LIN {X 0,Y 418.449,Z 234.861,A -85,B 0,C 180,E1 -9996.753,E2 -9996.753} C_VEL
LIN {X 0,Y 418.302,Z 234.881,A -85,B 0,C 180,E1 -9999.674,E2 -9999.674} C_VEL
LIN {X 0,Y 418.316,Z 234.874,A -85,B 0,C 180,E1 -10003.008,E2 -10003.008} C_VEL
LIN {X 0,Y 418.274,Z 234.878,A -85,B 0,C 180,E1 -10006.738,E2 -10006.738} C_VEL
LIN {X 0,Y 418.234,Z 234.89,A -85,B 0,C 180,E1 -10009.793,E2 -10009.793} C_VEL
LIN {X 0,Y 418.195,Z 234.888,A -85,B 0,C 180,E1 -10012.74,E2 -10012.74} C_VEL
LIN {X 0,Y 418.2,Z 234.893,A -85,B 0,C 180,E1 -10015.91,E2 -10015.91} C_VEL
LIN {X 0,Y 418.228,Z 234.884,A -85,B 0,C 180,E1 -10019.166,E2 -10019.166} C_VEL
LIN {X 0,Y 418.22,Z 234.886,A -85,B 0,C 180,E1 -10022.846,E2 -10022.846} C_VEL
LIN {X 0,Y 418.211,Z 234.892,A -85,B 0,C 180,E1 -10026.241,E2 -10026.241} C_VEL
LIN {X 0,Y 418.172,Z 234.891,A -85,B 0,C 180,E1 -10029.692,E2 -10029.692} C_VEL
LIN {X 0,Y 418.184,Z 234.894,A -85,B 0,C 180,E1 -10032.322,E2 -10032.322} C_VEL
LIN {X 0,Y 418.212,Z 234.889,A -85,B 0,C 180,E1 -10035.113,E2 -10035.113} C_VEL
LIN {X 0,Y 418.202,Z 234.887,A -85,B 0,C 180,E1 -10037.769,E2 -10037.769} C_VEL
LIN {X 0,Y 418.22,Z 234.886,A -85,B 0,C 180,E1 -10041.561,E2 -10041.561} C_VEL
LIN {X 0,Y 418.236,Z 234.889,A -85,B 0,C 180,E1 -10045.163,E2 -10045.163} C_VEL
LIN {X 0,Y 418.229,Z 234.887,A -85,B 0,C 180,E1 -10047.476,E2 -10047.476} C_VEL
LIN {X 0,Y 418.248,Z 234.885,A -85,B 0,C 180,E1 -10050.903,E2 -10050.903} C_VEL
LIN {X 0,Y 418.207,Z 234.887,A -85,B 0,C 180,E1 -10054.097,E2 -10054.097} C_VEL
LIN {X 0,Y 418.22,Z 234.891,A -85,B 0,C 180,E1 -10057.268,E2 -10057.268} C_VEL
LIN {X 0,Y 418.279,Z 234.878,A -85,B 0,C 180,E1 -10060.369,E2 -10060.369} C_VEL
LIN {X 0,Y 418.313,Z 234.878,A -85,B 0,C 180,E1 -10063.409,E2 -10063.409} C_VEL
LIN {X 0,Y 418.346,Z 234.87,A -85,B 0,C 180,E1 -10067.004,E2 -10067.004} C_VEL
LIN {X 0,Y 418.325,Z 234.874,A -85,B 0,C 180,E1 -10070.332,E2 -10070.332} C_VEL
LIN {X 0,Y 418.444,Z 234.858,A -85,B 0,C 180,E1 -10073.252,E2 -10073.252} C_VEL
LIN {X 0,Y 418.319,Z 234.873,A -85,B 0,C 180,E1 -10075.185,E2 -10075.185} C_VEL
LIN {X 0,Y 418.54,Z 234.853,A -85,B 0,C 180,E1 -10078.079,E2 -10078.079} C_VEL
LIN {X 0,Y 418.471,Z 234.854,A -85,B 0,C 180,E1 -10080.966,E2 -10080.966} C_VEL
LIN {X 0,Y 418.475,Z 234.854,A -85,B 0,C 180,E1 -10082.892,E2 -10082.892} C_VEL
LIN {X 0,Y 418.478,Z 234.854,A -85,B 0,C 180,E1 -10085.787,E2 -10085.787} C_VEL
LIN {X 0,Y 418.378,Z 234.87,A -85,B 0,C 180,E1 -10088.699,E2 -10088.699} C_VEL
LIN {X 0,Y 418.322,Z 234.872,A -85,B 0,C 180,E1 -10091.634,E2 -10091.634} C_VEL
LIN {X 0,Y 418.312,Z 234.881,A -85,B 0,C 180,E1 -10094.6,E2 -10094.6} C_VEL
LIN {X 0,Y 418.293,Z 234.876,A -85,B 0,C 180,E1 -10097.607,E2 -10097.607} C_VEL
LIN {X 0,Y 418.263,Z 234.885,A -85,B 0,C 180,E1 -10100.665,E2 -10100.665} C_VEL
LIN {X 0,Y 418.272,Z 234.878,A -85,B 0,C 180,E1 -10103.785,E2 -10103.785} C_VEL
LIN {X 0,Y 418.222,Z 234.893,A -85,B 0,C 180,E1 -10107.044,E2 -10107.044} C_VEL
LIN {X 0,Y 418.254,Z 234.881,A -85,B 0,C 180,E1 -10110.274,E2 -10110.274} C_VEL
LIN {X 0,Y 418.248,Z 234.884,A -85,B 0,C 180,E1 -10113.68,E2 -10113.68} C_VEL
LIN {X 0,Y 418.253,Z 234.887,A -85,B 0,C 180,E1 -10117.226,E2 -10117.226} C_VEL
LIN {X 0,Y 418.223,Z 234.886,A -85,B 0,C 180,E1 -10120.868,E2 -10120.868} C_VEL
LIN {X 0,Y 418.218,Z 234.891,A -85,B 0,C 180,E1 -10123.729,E2 -10123.729} C_VEL
LIN {X 0,Y 418.214,Z 234.886,A -85,B 0,C 180,E1 -10126.448,E2 -10126.448} C_VEL
LIN {X 0,Y 418.222,Z 234.886,A -85,B 0,C 180,E1 -10129.133,E2 -10129.133} C_VEL
LIN {X 0,Y 418.253,Z 234.881,A -85,B 0,C 180,E1 -10132.776,E2 -10132.776} C_VEL
LIN {X 0,Y 418.264,Z 234.883,A -85,B 0,C 180,E1 -10136.323,E2 -10136.323} C_VEL
LIN {X 0,Y 418.257,Z 234.883,A -85,B 0,C 180,E1 -10139.728,E2 -10139.728} C_VEL
LIN {X 0,Y 418.259,Z 234.887,A -85,B 0,C 180,E1 -10143.019,E2 -10143.019} C_VEL
LIN {X 0,Y 418.334,Z 234.998,A -85,B 0,C 180,E1 -10143.764,E2 -10143.764} C_VEL
LIN {X 0,Y 420.475,Z 246.2,A -85,B 0,C 180,E1 -10146.349,E2 -10146.349} C_VEL
LIN {X 0,Y 420.71,Z 251.116,A -85,B 0,C 180,E1 -10147.403,E2 -10147.403} C_VEL
LIN {X 0,Y 419.72,Z 266.974,A -85,B 0,C 180,E1 -10150.687,E2 -10150.687} C_VEL
LIN {X 0,Y 419.594,Z 269.57,A -85,B 0,C 180,E1 -10151.165,E2 -10151.165} C_VEL
LIN {X 0,Y 423.421,Z 293.744,A -85,B 0,C 180,E1 -10151.771,E2 -10151.771} C_VEL
LIN {X 0,Y 422.421,Z 377.284,A -85,B 0,C 180,E1 -10153.227,E2 -10153.227} C_VEL
LIN {X 0,Y 421.945,Z 390.495,A -85,B 0,C 180,E1 -10153.643,E2 -10153.643} C_VEL
LIN {X 0,Y 421.367,Z 403.772,A -85,B 0,C 180,E1 -10154.273,E2 -10154.273} C_VEL
LIN {X 0,Y 420.746,Z 414.923,A -85,B 0,C 180,E1 -10154.993,E2 -10154.993} C_VEL
LIN {X 0,Y 420.035,Z 426.239,A -85,B 0,C 180,E1 -10155.93,E2 -10155.93} C_VEL
LIN {X 0,Y 419.34,Z 436.982,A -85,B 0,C 180,E1 -10157.045,E2 -10157.045} C_VEL
LIN {X 0,Y 418.811,Z 445.521,A -85,B 0,C 180,E1 -10158.136,E2 -10158.136} C_VEL
LIN {X 0,Y 418.21,Z 453.382,A -85,B 0,C 180,E1 -10159.346,E2 -10159.346} C_VEL
LIN {X 0,Y 417.745,Z 461.051,A -85,B 0,C 180,E1 -10160.802,E2 -10160.802} C_VEL
LIN {X 0,Y 417.394,Z 467.211,A -85,B 0,C 180,E1 -10162.257,E2 -10162.257} C_VEL
LIN {X 0,Y 417.159,Z 472.14,A -85,B 0,C 180,E1 -10163.728,E2 -10163.728} C_VEL
LIN {X 0,Y 417.119,Z 475.84,A -85,B 0,C 180,E1 -10165.166,E2 -10165.166} C_VEL
LIN {X 0,Y 417.004,Z 477.771,A -85,B 0,C 180,E1 -10166.133,E2 -10166.133} C_VEL
LIN {X 0,Y 416.988,Z 479.275,A -85,B 0,C 180,E1 -10167.1,E2 -10167.1} C_VEL
LIN {X 0,Y 417.034,Z 480.328,A -85,B 0,C 180,E1 -10168.067,E2 -10168.067} C_VEL
LIN {X 0,Y 416.987,Z 481.263,A -85,B 0,C 180,E1 -10169.998,E2 -10169.998} C_VEL
LIN {X 0,Y 416.996,Z 481.142,A -85,B 0,C 180,E1 -10170.964,E2 -10170.964} C_VEL
LIN {X 0,Y 417.034,Z 480.589,A -85,B 0,C 180,E1 -10171.93,E2 -10171.93} C_VEL
LIN {X 0,Y 417.003,Z 478.309,A -85,B 0,C 180,E1 -10173.864,E2 -10173.864} C_VEL
LIN {X 0,Y 417.162,Z 475.485,A -85,B 0,C 180,E1 -10175.315,E2 -10175.315} C_VEL
LIN {X 0,Y 417.25,Z 471.64,A -85,B 0,C 180,E1 -10176.77,E2 -10176.77} C_VEL
LIN {X 0,Y 417.549,Z 466.675,A -85,B 0,C 180,E1 -10178.224,E2 -10178.224} C_VEL
LIN {X 0,Y 417.995,Z 460.442,A -85,B 0,C 180,E1 -10179.678,E2 -10179.678} C_VEL
LIN {X 0,Y 418.561,Z 452.662,A -85,B 0,C 180,E1 -10181.132,E2 -10181.132} C_VEL
LIN {X 0,Y 419.27,Z 444.726,A -85,B 0,C 180,E1 -10182.339,E2 -10182.339} C_VEL
LIN {X 0,Y 420.016,Z 435.055,A -85,B 0,C 180,E1 -10183.546,E2 -10183.546} C_VEL
LIN {X 0,Y 420.753,Z 424.328,A -85,B 0,C 180,E1 -10184.632,E2 -10184.632} C_VEL
LIN {X 0,Y 421.469,Z 413.916,A -85,B 0,C 180,E1 -10185.472,E2 -10185.472} C_VEL
LIN {X 0,Y 422.273,Z 401.439,A -85,B 0,C 180,E1 -10186.247,E2 -10186.247} C_VEL
LIN {X 0,Y 422.89,Z 388.32,A -85,B 0,C 180,E1 -10186.844,E2 -10186.844} C_VEL
LIN {X 0,Y 423.378,Z 376.495,A -85,B 0,C 180,E1 -10187.197,E2 -10187.197} C_VEL
LIN {X 0,Y 424.274,Z 292.712,A -85,B 0,C 180,E1 -10188.681,E2 -10188.681} C_VEL
LIN {X 0,Y 420.613,Z 272.268,A -85,B 0,C 180,E1 -10189.247,E2 -10189.247} C_VEL
LIN {X 0,Y 420.049,Z 269.214,A -85,B 0,C 180,E1 -10189.362,E2 -10189.362} C_VEL
LIN {X 0,Y 421.091,Z 253.587,A -85,B 0,C 180,E1 -10192.572,E2 -10192.572} C_VEL
LIN {X 0,Y 421.085,Z 248.782,A -85,B 0,C 180,E1 -10193.612,E2 -10193.612} C_VEL
LIN {X 0,Y 418.995,Z 238.02,A -85,B 0,C 180,E1 -10196.121,E2 -10196.121} C_VEL
LIN {X 0,Y 418.302,Z 234.921,A -85,B 0,C 180,E1 -10196.941,E2 -10196.941} C_VEL
LIN {X 0,Y 418.248,Z 234.885,A -85,B 0,C 180,E1 -10200.27,E2 -10200.27} C_VEL
LIN {X 0,Y 418.251,Z 234.886,A -85,B 0,C 180,E1 -10203.675,E2 -10203.675} C_VEL
LIN {X 0,Y 418.24,Z 234.886,A -85,B 0,C 180,E1 -10207.222,E2 -10207.222} C_VEL
LIN {X 0,Y 418.234,Z 234.886,A -85,B 0,C 180,E1 -10209.681,E2 -10209.681} C_VEL
LIN {X 0,Y 418.224,Z 234.882,A -85,B 0,C 180,E1 -10212.317,E2 -10212.317} C_VEL
LIN {X 0,Y 418.235,Z 234.883,A -85,B 0,C 180,E1 -10215.106,E2 -10215.106} C_VEL
LIN {X 0,Y 418.232,Z 234.879,A -85,B 0,C 180,E1 -10217.763,E2 -10217.763} C_VEL
LIN {X 0,Y 418.236,Z 234.884,A -85,B 0,C 180,E1 -10221.553,E2 -10221.553} C_VEL
LIN {X 0,Y 418.257,Z 234.884,A -85,B 0,C 180,E1 -10225.156,E2 -10225.156} C_VEL
LIN {X 0,Y 418.243,Z 234.881,A -85,B 0,C 180,E1 -10227.469,E2 -10227.469} C_VEL
LIN {X 0,Y 418.26,Z 234.882,A -85,B 0,C 180,E1 -10230.894,E2 -10230.894} C_VEL
LIN {X 0,Y 418.225,Z 234.885,A -85,B 0,C 180,E1 -10234.09,E2 -10234.09} C_VEL
LIN {X 0,Y 418.222,Z 234.888,A -85,B 0,C 180,E1 -10237.26,E2 -10237.26} C_VEL
LIN {X 0,Y 418.276,Z 234.878,A -85,B 0,C 180,E1 -10240.361,E2 -10240.361} C_VEL
LIN {X 0,Y 418.309,Z 234.874,A -85,B 0,C 180,E1 -10243.401,E2 -10243.401} C_VEL
LIN {X 0,Y 418.337,Z 234.873,A -85,B 0,C 180,E1 -10246.996,E2 -10246.996} C_VEL
LIN {X 0,Y 418.318,Z 234.874,A -85,B 0,C 180,E1 -10250.325,E2 -10250.325} C_VEL
LIN {X 0,Y 418.454,Z 234.856,A -85,B 0,C 180,E1 -10253.245,E2 -10253.245} C_VEL
LIN {X 0,Y 418.304,Z 234.881,A -85,B 0,C 180,E1 -10255.178,E2 -10255.178} C_VEL
LIN {X 0,Y 418.517,Z 234.85,A -85,B 0,C 180,E1 -10258.072,E2 -10258.072} C_VEL
LIN {X 0,Y 418.389,Z 234.864,A -85,B 0,C 180,E1 -10260.959,E2 -10260.959} C_VEL
LIN {X 0,Y 418.456,Z 234.856,A -85,B 0,C 180,E1 -10262.884,E2 -10262.884} C_VEL
LIN {X 0,Y 418.422,Z 234.86,A -85,B 0,C 180,E1 -10266.748,E2 -10266.748} C_VEL
LIN {X 0,Y 418.318,Z 234.874,A -85,B 0,C 180,E1 -10269.668,E2 -10269.668} C_VEL
LIN {X 0,Y 418.325,Z 234.87,A -85,B 0,C 180,E1 -10272.997,E2 -10272.997} C_VEL
LIN {X 0,Y 418.289,Z 234.876,A -85,B 0,C 180,E1 -10276.731,E2 -10276.731} C_VEL
LIN {X 0,Y 418.246,Z 234.885,A -85,B 0,C 180,E1 -10279.786,E2 -10279.786} C_VEL
LIN {X 0,Y 418.205,Z 234.889,A -85,B 0,C 180,E1 -10282.733,E2 -10282.733} C_VEL
LIN {X 0,Y 418.24,Z 234.885,A -85,B 0,C 180,E1 -10285.901,E2 -10285.901} C_VEL
LIN {X 0,Y 418.235,Z 234.88,A -85,B 0,C 180,E1 -10289.159,E2 -10289.159} C_VEL
LIN {X 0,Y 418.226,Z 234.884,A -85,B 0,C 180,E1 -10292.841,E2 -10292.841} C_VEL
LIN {X 0,Y 418.216,Z 234.886,A -85,B 0,C 180,E1 -10296.236,E2 -10296.236} C_VEL
LIN {X 0,Y 418.232,Z 234.888,A -85,B 0,C 180,E1 -10299.677,E2 -10299.677} C_VEL
LIN {X 0,Y 418.249,Z 234.885,A -85,B 0,C 180,E1 -10302.327,E2 -10302.327} C_VEL
LIN {X 0,Y 418.289,Z 234.973,A -85,B 0,C 180,E1 -10304.337,E2 -10304.337} C_VEL
LIN {X 0,Y 419.722,Z 241.882,A -85,B 0,C 180,E1 -10306.048,E2 -10306.048} C_VEL
LIN {X 0,Y 420.664,Z 247.281,A -85,B 0,C 180,E1 -10307.308,E2 -10307.308} C_VEL
LIN {X 0,Y 420.284,Z 256.46,A -85,B 0,C 180,E1 -10309.298,E2 -10309.298} C_VEL
LIN {X 0,Y 420.229,Z 258.615,A -85,B 0,C 180,E1 -10309.697,E2 -10309.697} C_VEL
LIN {X 0,Y 424.167,Z 278.047,A -85,B 0,C 180,E1 -10310.287,E2 -10310.287} C_VEL
LIN {X 0,Y 424.537,Z 281.534,A -85,B 0,C 180,E1 -10310.369,E2 -10310.369} C_VEL
LIN {X 0,Y 423.399,Z 365.98,A -85,B 0,C 180,E1 -10311.858,E2 -10311.858} C_VEL
LIN {X 0,Y 422.926,Z 379.212,A -85,B 0,C 180,E1 -10312.279,E2 -10312.279} C_VEL
LIN {X 0,Y 422.339,Z 391.655,A -85,B 0,C 180,E1 -10312.868,E2 -10312.868} C_VEL
LIN {X 0,Y 421.708,Z 402.839,A -85,B 0,C 180,E1 -10313.581,E2 -10313.581} C_VEL
LIN {X 0,Y 420.896,Z 414.682,A -85,B 0,C 180,E1 -10314.562,E2 -10314.562} C_VEL
LIN {X 0,Y 420.119,Z 424.963,A -85,B 0,C 180,E1 -10315.628,E2 -10315.628} C_VEL
LIN {X 0,Y 419.404,Z 433.62,A -85,B 0,C 180,E1 -10316.727,E2 -10316.727} C_VEL
LIN {X 0,Y 418.702,Z 442.352,A -85,B 0,C 180,E1 -10318.082,E2 -10318.082} C_VEL
LIN {X 0,Y 418.028,Z 450.685,A -85,B 0,C 180,E1 -10319.713,E2 -10319.713} C_VEL
LIN {X 0,Y 417.741,Z 456.001,A -85,B 0,C 180,E1 -10321.014,E2 -10321.014} C_VEL
LIN {X 0,Y 417.405,Z 460.637,A -85,B 0,C 180,E1 -10322.419,E2 -10322.419} C_VEL
LIN {X 0,Y 417.16,Z 464.674,A -85,B 0,C 180,E1 -10324.024,E2 -10324.024} C_VEL
LIN {X 0,Y 416.946,Z 467.333,A -85,B 0,C 180,E1 -10325.522,E2 -10325.522} C_VEL
LIN {X 0,Y 416.8,Z 469.126,A -85,B 0,C 180,E1 -10327.183,E2 -10327.183} C_VEL
LIN {X 0,Y 416.823,Z 469.641,A -85,B 0,C 180,E1 -10328.228,E2 -10328.228} C_VEL
LIN {X 0,Y 416.779,Z 469.681,A -85,B 0,C 180,E1 -10329.263,E2 -10329.263} C_VEL
LIN {X 0,Y 416.874,Z 468.974,A -85,B 0,C 180,E1 -10330.733,E2 -10330.733} C_VEL
LIN {X 0,Y 416.903,Z 467.138,A -85,B 0,C 180,E1 -10332.338,E2 -10332.338} C_VEL
LIN {X 0,Y 417.086,Z 464.431,A -85,B 0,C 180,E1 -10333.813,E2 -10333.813} C_VEL
LIN {X 0,Y 417.278,Z 460.442,A -85,B 0,C 180,E1 -10335.368,E2 -10335.368} C_VEL
LIN {X 0,Y 417.558,Z 455.374,A -85,B 0,C 180,E1 -10336.868,E2 -10336.868} C_VEL
LIN {X 0,Y 417.962,Z 448.983,A -85,B 0,C 180,E1 -10338.361,E2 -10338.361} C_VEL
LIN {X 0,Y 418.45,Z 440.984,A -85,B 0,C 180,E1 -10339.844,E2 -10339.844} C_VEL
LIN {X 0,Y 419.056,Z 432.78,A -85,B 0,C 180,E1 -10341.077,E2 -10341.077} C_VEL
LIN {X 0,Y 419.673,Z 422.808,A -85,B 0,C 180,E1 -10342.302,E2 -10342.302} C_VEL
LIN {X 0,Y 419.733,Z 422.251,A -85,B 0,C 180,E1 -10342.364,E2 -10342.364} C_VEL
LIN {X 0,Y 419.504,Z 417.637,A -85,B 0,C 180,E1 -10342.867,E2 -10342.867} C_VEL
LIN {X 0,Y 417.189,Z 409.926,A -85,B 0,C 180,E1 -10343.663,E2 -10343.663} C_VEL
LIN {X 0,Y 414.801,Z 401.806,A -85,B 0,C 180,E1 -10344.38,E2 -10344.38} C_VEL
LIN {X 0,Y 414.451,Z 396.549,A -85,B 0,C 180,E1 -10344.75,E2 -10344.75} C_VEL
LIN {X 0,Y 414.994,Z 384.483,A -85,B 0,C 180,E1 -10345.412,E2 -10345.412} C_VEL
LIN {X 0,Y 415.503,Z 371.242,A -85,B 0,C 180,E1 -10345.922,E2 -10345.922} C_VEL
LIN {X 0,Y 415.745,Z 357.284,A -85,B 0,C 180,E1 -10346.239,E2 -10346.239} C_VEL
LIN {X 0,Y 416.51,Z 280.026,A -85,B 0,C 180,E1 -10347.584,E2 -10347.584} C_VEL
LIN {X 0,Y 412.836,Z 258.965,A -85,B 0,C 180,E1 -10348.142,E2 -10348.142} C_VEL
LIN {X 0,Y 412.957,Z 255.755,A -85,B 0,C 180,E1 -10348.783,E2 -10348.783} C_VEL
LIN {X 0,Y 413.419,Z 247.118,A -85,B 0,C 180,E1 -10350.732,E2 -10350.732} C_VEL
LIN {X 0,Y 411.82,Z 238.008,A -85,B 0,C 180,E1 -10352.936,E2 -10352.936} C_VEL
LIN {X 0,Y 411.281,Z 235.803,A -85,B 0,C 180,E1 -10353.553,E2 -10353.553} C_VEL
LIN {X 0,Y 411.431,Z 235.736,A -85,B 0,C 180,E1 -10355.884,E2 -10355.884} C_VEL
LIN {X 0,Y 411.314,Z 235.746,A -85,B 0,C 180,E1 -10358.848,E2 -10358.848} C_VEL
LIN {X 0,Y 411.258,Z 235.757,A -85,B 0,C 180,E1 -10361.835,E2 -10361.835} C_VEL
LIN {X 0,Y 411.222,Z 235.757,A -85,B 0,C 180,E1 -10364.855,E2 -10364.855} C_VEL
LIN {X 0,Y 411.214,Z 235.764,A -85,B 0,C 180,E1 -10367.918,E2 -10367.918} C_VEL
LIN {X 0,Y 411.16,Z 235.764,A -85,B 0,C 180,E1 -10371.037,E2 -10371.037} C_VEL
LIN {X 0,Y 411.168,Z 235.768,A -85,B 0,C 180,E1 -10374.22,E2 -10374.22} C_VEL
LIN {X 0,Y 411.154,Z 235.766,A -85,B 0,C 180,E1 -10377.487,E2 -10377.487} C_VEL
LIN {X 0,Y 411.157,Z 235.766,A -85,B 0,C 180,E1 -10380.852,E2 -10380.852} C_VEL
LIN {X 0,Y 411.163,Z 235.772,A -85,B 0,C 180,E1 -10384.339,E2 -10384.339} C_VEL
LIN {X 0,Y 411.158,Z 235.768,A -85,B 0,C 180,E1 -10386.747,E2 -10386.747} C_VEL
LIN {X 0,Y 411.141,Z 235.767,A -85,B 0,C 180,E1 -10389.724,E2 -10389.724} C_VEL
LIN {X 0,Y 411.139,Z 235.769,A -85,B 0,C 180,E1 -10393.14,E2 -10393.14} C_VEL
LIN {X 0,Y 411.142,Z 235.767,A -85,B 0,C 180,E1 -10395.886,E2 -10395.886} C_VEL
LIN {X 0,Y 411.13,Z 235.776,A -85,B 0,C 180,E1 -10398.779,E2 -10398.779} C_VEL
LIN {X 0,Y 411.169,Z 235.763,A -85,B 0,C 180,E1 -10402.03,E2 -10402.03} C_VEL
LIN {X 0,Y 411.188,Z 235.767,A -85,B 0,C 180,E1 -10405.128,E2 -10405.128} C_VEL
LIN {X 0,Y 411.149,Z 235.766,A -85,B 0,C 180,E1 -10408.007,E2 -10408.007} C_VEL
LIN {X 0,Y 411.161,Z 235.77,A -85,B 0,C 180,E1 -10411.411,E2 -10411.411} C_VEL
LIN {X 0,Y 411.179,Z 235.765,A -85,B 0,C 180,E1 -10414.946,E2 -10414.946} C_VEL
LIN {X 0,Y 411.197,Z 235.762,A -85,B 0,C 180,E1 -10417.918,E2 -10417.918} C_VEL
LIN {X 0,Y 411.214,Z 235.76,A -85,B 0,C 180,E1 -10421.056,E2 -10421.056} C_VEL
LIN {X 0,Y 411.248,Z 235.755,A -85,B 0,C 180,E1 -10424.136,E2 -10424.136} C_VEL
LIN {X 0,Y 411.302,Z 235.748,A -85,B 0,C 180,E1 -10427.17,E2 -10427.17} C_VEL
LIN {X 0,Y 411.279,Z 235.753,A -85,B 0,C 180,E1 -10430.165,E2 -10430.165} C_VEL
LIN {X 0,Y 411.393,Z 235.736,A -85,B 0,C 180,E1 -10433.136,E2 -10433.136} C_VEL
LIN {X 0,Y 411.29,Z 235.748,A -85,B 0,C 180,E1 -10435.103,E2 -10435.103} C_VEL
LIN {X 0,Y 411.508,Z 235.728,A -85,B 0,C 180,E1 -10438.046,E2 -10438.046} C_VEL
LIN {X 0,Y 411.436,Z 235.73,A -85,B 0,C 180,E1 -10440.983,E2 -10440.983} C_VEL
LIN {X 0,Y 411.433,Z 235.731,A -85,B 0,C 180,E1 -10442.941,E2 -10442.941} C_VEL
LIN {X 0,Y 411.4,Z 235.737,A -85,B 0,C 180,E1 -10446.872,E2 -10446.872} C_VEL
LIN {X 0,Y 411.291,Z 235.749,A -85,B 0,C 180,E1 -10449.842,E2 -10449.842} C_VEL
LIN {X 0,Y 411.318,Z 235.746,A -85,B 0,C 180,E1 -10453.107,E2 -10453.107} C_VEL
LIN {X 0,Y 411.271,Z 235.756,A -85,B 0,C 180,E1 -10456.891,E2 -10456.891} C_VEL
LIN {X 0,Y 411.245,Z 235.754,A -85,B 0,C 180,E1 -10459.989,E2 -10459.989} C_VEL
LIN {X 0,Y 411.202,Z 235.764,A -85,B 0,C 180,E1 -10463.151,E2 -10463.151} C_VEL
LIN {X 0,Y 411.19,Z 235.762,A -85,B 0,C 180,E1 -10466.387,E2 -10466.387} C_VEL
LIN {X 0,Y 411.21,Z 235.759,A -85,B 0,C 180,E1 -10469.715,E2 -10469.715} C_VEL
LIN {X 0,Y 411.22,Z 235.764,A -85,B 0,C 180,E1 -10473.158,E2 -10473.158} C_VEL
LIN {X 0,Y 411.207,Z 235.759,A -85,B 0,C 180,E1 -10476.553,E2 -10476.553} C_VEL
LIN {X 0,Y 411.185,Z 235.766,A -85,B 0,C 180,E1 -10479.721,E2 -10479.721} C_VEL
LIN {X 0,Y 411.178,Z 235.765,A -85,B 0,C 180,E1 -10483.136,E2 -10483.136} C_VEL
LIN {X 0,Y 411.178,Z 235.767,A -85,B 0,C 180,E1 -10485.883,E2 -10485.883} C_VEL
LIN {X 0,Y 411.162,Z 235.764,A -85,B 0,C 180,E1 -10488.775,E2 -10488.775} C_VEL
LIN {X 0,Y 411.201,Z 235.765,A -85,B 0,C 180,E1 -10492.025,E2 -10492.025} C_VEL
LIN {X 0,Y 411.221,Z 235.761,A -85,B 0,C 180,E1 -10495.666,E2 -10495.666} C_VEL
LIN {X 0,Y 411.204,Z 235.761,A -85,B 0,C 180,E1 -10499.152,E2 -10499.152} C_VEL
LIN {X 0,Y 411.203,Z 235.764,A -85,B 0,C 180,E1 -10502.517,E2 -10502.517} C_VEL
LIN {X 0,Y 411.282,Z 235.896,A -85,B 0,C 180,E1 -10503.554,E2 -10503.554} C_VEL
LIN {X 0,Y 413.537,Z 247.629,A -85,B 0,C 180,E1 -10506.304,E2 -10506.304} C_VEL
LIN {X 0,Y 413.76,Z 252.034,A -85,B 0,C 180,E1 -10507.266,E2 -10507.266} C_VEL
LIN {X 0,Y 412.651,Z 268.883,A -85,B 0,C 180,E1 -10510.795,E2 -10510.795} C_VEL
LIN {X 0,Y 412.738,Z 270.227,A -85,B 0,C 180,E1 -10510.913,E2 -10510.913} C_VEL
LIN {X 0,Y 416.598,Z 295.2,A -85,B 0,C 180,E1 -10511.529,E2 -10511.529} C_VEL
LIN {X 0,Y 415.571,Z 377.135,A -85,B 0,C 180,E1 -10512.974,E2 -10512.974} C_VEL
LIN {X 0,Y 415.098,Z 390.362,A -85,B 0,C 180,E1 -10513.397,E2 -10513.397} C_VEL
LIN {X 0,Y 414.528,Z 403.095,A -85,B 0,C 180,E1 -10514.006,E2 -10514.006} C_VEL
LIN {X 0,Y 413.857,Z 414.407,A -85,B 0,C 180,E1 -10514.738,E2 -10514.738} C_VEL
LIN {X 0,Y 413.066,Z 426.401,A -85,B 0,C 180,E1 -10515.746,E2 -10515.746} C_VEL
LIN {X 0,Y 412.386,Z 436.603,A -85,B 0,C 180,E1 -10516.823,E2 -10516.823} C_VEL
LIN {X 0,Y 411.805,Z 445.188,A -85,B 0,C 180,E1 -10517.931,E2 -10517.931} C_VEL
LIN {X 0,Y 411.19,Z 453.095,A -85,B 0,C 180,E1 -10519.162,E2 -10519.162} C_VEL
LIN {X 0,Y 410.692,Z 460.807,A -85,B 0,C 180,E1 -10520.642,E2 -10520.642} C_VEL
LIN {X 0,Y 410.348,Z 466.996,A -85,B 0,C 180,E1 -10522.123,E2 -10522.123} C_VEL
LIN {X 0,Y 410.057,Z 472.387,A -85,B 0,C 180,E1 -10523.77,E2 -10523.77} C_VEL
LIN {X 0,Y 410.033,Z 475.674,A -85,B 0,C 180,E1 -10525.082,E2 -10525.082} C_VEL
LIN {X 0,Y 409.924,Z 477.616,A -85,B 0,C 180,E1 -10526.066,E2 -10526.066} C_VEL
LIN {X 0,Y 409.886,Z 479.137,A -85,B 0,C 180,E1 -10527.05,E2 -10527.05} C_VEL
LIN {X 0,Y 409.93,Z 480.204,A -85,B 0,C 180,E1 -10528.034,E2 -10528.034} C_VEL
LIN {X 0,Y 409.922,Z 480.875,A -85,B 0,C 180,E1 -10529.016,E2 -10529.016} C_VEL
LIN {X 0,Y 409.91,Z 481.159,A -85,B 0,C 180,E1 -10529.998,E2 -10529.998} C_VEL
LIN {X 0,Y 409.922,Z 481.053,A -85,B 0,C 180,E1 -10530.981,E2 -10530.981} C_VEL
LIN {X 0,Y 409.93,Z 480.515,A -85,B 0,C 180,E1 -10531.963,E2 -10531.963} C_VEL
LIN {X 0,Y 409.925,Z 478.254,A -85,B 0,C 180,E1 -10533.931,E2 -10533.931} C_VEL
LIN {X 0,Y 410.08,Z 475.45,A -85,B 0,C 180,E1 -10535.407,E2 -10535.407} C_VEL
LIN {X 0,Y 410.188,Z 471.625,A -85,B 0,C 180,E1 -10536.887,E2 -10536.887} C_VEL
LIN {X 0,Y 410.498,Z 466.683,A -85,B 0,C 180,E1 -10538.366,E2 -10538.366} C_VEL
LIN {X 0,Y 410.969,Z 460.473,A -85,B 0,C 180,E1 -10539.845,E2 -10539.845} C_VEL
LIN {X 0,Y 411.562,Z 452.748,A -85,B 0,C 180,E1 -10541.324,E2 -10541.324} C_VEL
LIN {X 0,Y 412.46,Z 443.089,A -85,B 0,C 180,E1 -10542.796,E2 -10542.796} C_VEL
LIN {X 0,Y 413.312,Z 432.87,A -85,B 0,C 180,E1 -10544.051,E2 -10544.051} C_VEL
LIN {X 0,Y 414.107,Z 421.887,A -85,B 0,C 180,E1 -10545.124,E2 -10545.124} C_VEL
LIN {X 0,Y 414.879,Z 410.892,A -85,B 0,C 180,E1 -10545.977,E2 -10545.977} C_VEL
LIN {X 0,Y 415.754,Z 398.708,A -85,B 0,C 180,E1 -10546.699,E2 -10546.699} C_VEL
LIN {X 0,Y 416.313,Z 385.939,A -85,B 0,C 180,E1 -10547.245,E2 -10547.245} C_VEL
LIN {X 0,Y 416.776,Z 372.494,A -85,B 0,C 180,E1 -10547.605,E2 -10547.605} C_VEL
LIN {X 0,Y 417.675,Z 293.704,A -85,B 0,C 180,E1 -10549.01,E2 -10549.01} C_VEL
LIN {X 0,Y 414.142,Z 273.998,A -85,B 0,C 180,E1 -10549.57,E2 -10549.57} C_VEL
LIN {X 0,Y 413.187,Z 269.043,A -85,B 0,C 180,E1 -10549.749,E2 -10549.749} C_VEL
LIN {X 0,Y 414.184,Z 254.928,A -85,B 0,C 180,E1 -10552.706,E2 -10552.706} C_VEL
LIN {X 0,Y 414.264,Z 250.697,A -85,B 0,C 180,E1 -10553.632,E2 -10553.632} C_VEL
LIN {X 0,Y 412.025,Z 239.366,A -85,B 0,C 180,E1 -10556.325,E2 -10556.325} C_VEL
LIN {X 0,Y 411.268,Z 235.805,A -85,B 0,C 180,E1 -10557.268,E2 -10557.268} C_VEL
LIN {X 0,Y 411.205,Z 235.768,A -85,B 0,C 180,E1 -10559.71,E2 -10559.71} C_VEL
LIN {X 0,Y 411.211,Z 235.759,A -85,B 0,C 180,E1 -10563.153,E2 -10563.153} C_VEL
LIN {X 0,Y 411.194,Z 235.765,A -85,B 0,C 180,E1 -10566.549,E2 -10566.549} C_VEL
LIN {X 0,Y 411.2,Z 235.763,A -85,B 0,C 180,E1 -10569.722,E2 -10569.722} C_VEL
LIN {X 0,Y 411.171,Z 235.763,A -85,B 0,C 180,E1 -10573.131,E2 -10573.131} C_VEL
LIN {X 0,Y 411.167,Z 235.761,A -85,B 0,C 180,E1 -10575.879,E2 -10575.879} C_VEL
LIN {X 0,Y 411.152,Z 235.771,A -85,B 0,C 180,E1 -10578.771,E2 -10578.771} C_VEL
LIN {X 0,Y 411.184,Z 235.765,A -85,B 0,C 180,E1 -10582.022,E2 -10582.022} C_VEL
LIN {X 0,Y 411.203,Z 235.761,A -85,B 0,C 180,E1 -10585.663,E2 -10585.663} C_VEL
LIN {X 0,Y 411.186,Z 235.764,A -85,B 0,C 180,E1 -10589.149,E2 -10589.149} C_VEL
LIN {X 0,Y 411.179,Z 235.763,A -85,B 0,C 180,E1 -10591.404,E2 -10591.404} C_VEL
LIN {X 0,Y 411.207,Z 235.76,A -85,B 0,C 180,E1 -10594.931,E2 -10594.931} C_VEL
LIN {X 0,Y 411.197,Z 235.759,A -85,B 0,C 180,E1 -10597.91,E2 -10597.91} C_VEL
LIN {X 0,Y 411.212,Z 235.765,A -85,B 0,C 180,E1 -10601.048,E2 -10601.048} C_VEL
LIN {X 0,Y 411.244,Z 235.752,A -85,B 0,C 180,E1 -10604.128,E2 -10604.128} C_VEL
LIN {X 0,Y 411.294,Z 235.748,A -85,B 0,C 180,E1 -10607.162,E2 -10607.162} C_VEL
LIN {X 0,Y 411.271,Z 235.752,A -85,B 0,C 180,E1 -10610.157,E2 -10610.157} C_VEL
LIN {X 0,Y 411.42,Z 235.73,A -85,B 0,C 180,E1 -10613.129,E2 -10613.129} C_VEL
LIN {X 0,Y 411.277,Z 235.755,A -85,B 0,C 180,E1 -10615.095,E2 -10615.095} C_VEL
LIN {X 0,Y 411.486,Z 235.726,A -85,B 0,C 180,E1 -10618.039,E2 -10618.039} C_VEL
LIN {X 0,Y 411.487,Z 235.727,A -85,B 0,C 180,E1 -10621.954,E2 -10621.954} C_VEL
LIN {X 0,Y 411.367,Z 235.738,A -85,B 0,C 180,E1 -10626.479,E2 -10626.479} C_VEL
LIN {X 0,Y 411.299,Z 235.746,A -85,B 0,C 180,E1 -10628.842,E2 -10628.842} C_VEL
LIN {X 0,Y 411.262,Z 235.758,A -85,B 0,C 180,E1 -10631.829,E2 -10631.829} C_VEL
LIN {X 0,Y 411.236,Z 235.757,A -85,B 0,C 180,E1 -10634.849,E2 -10634.849} C_VEL
LIN {X 0,Y 411.221,Z 235.762,A -85,B 0,C 180,E1 -10637.912,E2 -10637.912} C_VEL
LIN {X 0,Y 411.171,Z 235.765,A -85,B 0,C 180,E1 -10641.031,E2 -10641.031} C_VEL
LIN {X 0,Y 411.193,Z 235.767,A -85,B 0,C 180,E1 -10644.212,E2 -10644.212} C_VEL
LIN {X 0,Y 411.23,Z 235.757,A -85,B 0,C 180,E1 -10647.474,E2 -10647.474} C_VEL
LIN {X 0,Y 411.159,Z 235.769,A -85,B 0,C 180,E1 -10650.844,E2 -10650.844} C_VEL
LIN {X 0,Y 411.175,Z 235.77,A -85,B 0,C 180,E1 -10654.33,E2 -10654.33} C_VEL
LIN {X 0,Y 411.171,Z 235.766,A -85,B 0,C 180,E1 -10657.97,E2 -10657.97} C_VEL
LIN {X 0,Y 411.175,Z 235.77,A -85,B 0,C 180,E1 -10661.233,E2 -10661.233} C_VEL
LIN {X 0,Y 411.261,Z 235.913,A -85,B 0,C 180,E1 -10664.047,E2 -10664.047} C_VEL
LIN {X 0,Y 413.371,Z 246.305,A -85,B 0,C 180,E1 -10666.612,E2 -10666.612} C_VEL
LIN {X 0,Y 413.815,Z 250.306,A -85,B 0,C 180,E1 -10667.542,E2 -10667.542} C_VEL
LIN {X 0,Y 413.365,Z 258.584,A -85,B 0,C 180,E1 -10669.299,E2 -10669.299} C_VEL
LIN {X 0,Y 415.393,Z 267.942,A -85,B 0,C 180,E1 -10669.626,E2 -10669.626} C_VEL
LIN {X 0,Y 417.925,Z 281.248,A -85,B 0,C 180,E1 -10670.012,E2 -10670.012} C_VEL
LIN {X 0,Y 416.703,Z 366.578,A -85,B 0,C 180,E1 -10671.546,E2 -10671.546} C_VEL
LIN {X 0,Y 416.195,Z 380.084,A -85,B 0,C 180,E1 -10671.991,E2 -10671.991} C_VEL
LIN {X 0,Y 415.566,Z 393.064,A -85,B 0,C 180,E1 -10672.633,E2 -10672.633} C_VEL
LIN {X 0,Y 414.769,Z 405.479,A -85,B 0,C 180,E1 -10673.477,E2 -10673.477} C_VEL
LIN {X 0,Y 413.911,Z 416.416,A -85,B 0,C 180,E1 -10674.431,E2 -10674.431} C_VEL
LIN {X 0,Y 413.127,Z 426.7,A -85,B 0,C 180,E1 -10675.556,E2 -10675.556} C_VEL
LIN {X 0,Y 412.39,Z 435.254,A -85,B 0,C 180,E1 -10676.703,E2 -10676.703} C_VEL
LIN {X 0,Y 411.667,Z 443.474,A -85,B 0,C 180,E1 -10678.048,E2 -10678.048} C_VEL
LIN {X 0,Y 410.98,Z 451.612,A -85,B 0,C 180,E1 -10679.706,E2 -10679.706} C_VEL
LIN {X 0,Y 410.578,Z 457.912,A -85,B 0,C 180,E1 -10681.363,E2 -10681.363} C_VEL
LIN {X 0,Y 410.247,Z 462.593,A -85,B 0,C 180,E1 -10682.963,E2 -10682.963} C_VEL
LIN {X 0,Y 410.007,Z 466.156,A -85,B 0,C 180,E1 -10684.628,E2 -10684.628} C_VEL
LIN {X 0,Y 409.836,Z 467.818,A -85,B 0,C 180,E1 -10685.699,E2 -10685.699} C_VEL
LIN {X 0,Y 409.743,Z 468.939,A -85,B 0,C 180,E1 -10686.767,E2 -10686.767} C_VEL
LIN {X 0,Y 409.705,Z 469.622,A -85,B 0,C 180,E1 -10687.85,E2 -10687.85} C_VEL
LIN {X 0,Y 409.693,Z 469.837,A -85,B 0,C 180,E1 -10688.887,E2 -10688.887} C_VEL
LIN {X 0,Y 409.773,Z 469.184,A -85,B 0,C 180,E1 -10690.596,E2 -10690.596} C_VEL
LIN {X 0,Y 409.778,Z 467.742,A -85,B 0,C 180,E1 -10692.02,E2 -10692.02} C_VEL
LIN {X 0,Y 409.979,Z 464.859,A -85,B 0,C 180,E1 -10693.712,E2 -10693.712} C_VEL
LIN {X 0,Y 410.156,Z 461.519,A -85,B 0,C 180,E1 -10695.108,E2 -10695.108} C_VEL
LIN {X 0,Y 410.434,Z 456.707,A -85,B 0,C 180,E1 -10696.636,E2 -10696.636} C_VEL
LIN {X 0,Y 410.787,Z 450.607,A -85,B 0,C 180,E1 -10698.154,E2 -10698.154} C_VEL
LIN {X 0,Y 411.281,Z 443.002,A -85,B 0,C 180,E1 -10699.665,E2 -10699.665} C_VEL
LIN {X 0,Y 411.915,Z 435.208,A -85,B 0,C 180,E1 -10700.921,E2 -10700.921} C_VEL
LIN {X 0,Y 412.545,Z 425.768,A -85,B 0,C 180,E1 -10702.169,E2 -10702.169} C_VEL
LIN {X 0,Y 413.335,Z 415.185,A -85,B 0,C 180,E1 -10703.289,E2 -10703.289} C_VEL
LIN {X 0,Y 414.058,Z 403.46,A -85,B 0,C 180,E1 -10704.279,E2 -10704.279} C_VEL
LIN {X 0,Y 414.451,Z 396.549,A -85,B 0,C 180,E1 -10704.75,E2 -10704.75} C_VEL
LIN {X 0,Y 414.131,Z 391.214,A -85,B 0,C 180,E1 -10705.089,E2 -10705.089} C_VEL
LIN {X 0,Y 411.783,Z 382.369,A -85,B 0,C 180,E1 -10705.628,E2 -10705.628} C_VEL
LIN {X 0,Y 409.293,Z 373.334,A -85,B 0,C 180,E1 -10706.077,E2 -10706.077} C_VEL
LIN {X 0,Y 408.733,Z 367.626,A -85,B 0,C 180,E1 -10706.272,E2 -10706.272} C_VEL
LIN {X 0,Y 409.146,Z 335.693,A -85,B 0,C 180,E1 -10706.877,E2 -10706.877} C_VEL
LIN {X 0,Y 409.76,Z 281.107,A -85,B 0,C 180,E1 -10707.843,E2 -10707.843} C_VEL
LIN {X 0,Y 405.884,Z 258.981,A -85,B 0,C 180,E1 -10708.445,E2 -10708.445} C_VEL
LIN {X 0,Y 406.271,Z 252.937,A -85,B 0,C 180,E1 -10709.754,E2 -10709.754} C_VEL
LIN {X 0,Y 406.37,Z 247.602,A -85,B 0,C 180,E1 -10710.992,E2 -10710.992} C_VEL
LIN {X 0,Y 404.885,Z 239.512,A -85,B 0,C 180,E1 -10712.986,E2 -10712.986} C_VEL
LIN {X 0,Y 404.208,Z 236.669,A -85,B 0,C 180,E1 -10713.771,E2 -10713.771} C_VEL
LIN {X 0,Y 404.379,Z 236.615,A -85,B 0,C 180,E1 -10715.987,E2 -10715.987} C_VEL
LIN {X 0,Y 404.251,Z 236.627,A -85,B 0,C 180,E1 -10719.003,E2 -10719.003} C_VEL
LIN {X 0,Y 404.229,Z 236.63,A -85,B 0,C 180,E1 -10722.044,E2 -10722.044} C_VEL
LIN {X 0,Y 404.168,Z 236.637,A -85,B 0,C 180,E1 -10725.121,E2 -10725.121} C_VEL
LIN {X 0,Y 404.172,Z 236.638,A -85,B 0,C 180,E1 -10728.241,E2 -10728.241} C_VEL
LIN {X 0,Y 404.102,Z 236.646,A -85,B 0,C 180,E1 -10731.423,E2 -10731.423} C_VEL
LIN {X 0,Y 404.126,Z 236.642,A -85,B 0,C 180,E1 -10734.67,E2 -10734.67} C_VEL
LIN {X 0,Y 404.096,Z 236.65,A -85,B 0,C 180,E1 -10738.009,E2 -10738.009} C_VEL
LIN {X 0,Y 404.112,Z 236.649,A -85,B 0,C 180,E1 -10740.289,E2 -10740.289} C_VEL
LIN {X 0,Y 404.108,Z 236.645,A -85,B 0,C 180,E1 -10743.817,E2 -10743.817} C_VEL
LIN {X 0,Y 404.103,Z 236.646,A -85,B 0,C 180,E1 -10746.878,E2 -10746.878} C_VEL
LIN {X 0,Y 404.092,Z 236.647,A -85,B 0,C 180,E1 -10750.079,E2 -10750.079} C_VEL
LIN {X 0,Y 404.118,Z 236.644,A -85,B 0,C 180,E1 -10753.086,E2 -10753.086} C_VEL
LIN {X 0,Y 404.123,Z 236.641,A -85,B 0,C 180,E1 -10755.93,E2 -10755.93} C_VEL
LIN {X 0,Y 404.084,Z 236.651,A -85,B 0,C 180,E1 -10758.638,E2 -10758.638} C_VEL
LIN {X 0,Y 404.123,Z 236.642,A -85,B 0,C 180,E1 -10761.5,E2 -10761.5} C_VEL
LIN {X 0,Y 404.159,Z 236.644,A -85,B 0,C 180,E1 -10764.988,E2 -10764.988} C_VEL
LIN {X 0,Y 404.124,Z 236.642,A -85,B 0,C 180,E1 -10768.448,E2 -10768.448} C_VEL
LIN {X 0,Y 404.138,Z 236.643,A -85,B 0,C 180,E1 -10770.867,E2 -10770.867} C_VEL
LIN {X 0,Y 404.144,Z 236.64,A -85,B 0,C 180,E1 -10774.728,E2 -10774.728} C_VEL
LIN {X 0,Y 404.16,Z 236.643,A -85,B 0,C 180,E1 -10777.513,E2 -10777.513} C_VEL
LIN {X 0,Y 404.158,Z 236.637,A -85,B 0,C 180,E1 -10780.712,E2 -10780.712} C_VEL
LIN {X 0,Y 404.217,Z 236.634,A -85,B 0,C 180,E1 -10783.853,E2 -10783.853} C_VEL
LIN {X 0,Y 404.284,Z 236.621,A -85,B 0,C 180,E1 -10786.943,E2 -10786.943} C_VEL
LIN {X 0,Y 404.246,Z 236.631,A -85,B 0,C 180,E1 -10789.992,E2 -10789.992} C_VEL
LIN {X 0,Y 404.344,Z 236.613,A -85,B 0,C 180,E1 -10793.016,E2 -10793.016} C_VEL
LIN {X 0,Y 404.261,Z 236.624,A -85,B 0,C 180,E1 -10795.017,E2 -10795.017} C_VEL
LIN {X 0,Y 404.477,Z 236.604,A -85,B 0,C 180,E1 -10798.012,E2 -10798.012} C_VEL
LIN {X 0,Y 404.402,Z 236.606,A -85,B 0,C 180,E1 -10801,E2 -10801} C_VEL
LIN {X 0,Y 404.367,Z 236.611,A -85,B 0,C 180,E1 -10802.993,E2 -10802.993} C_VEL
LIN {X 0,Y 404.376,Z 236.613,A -85,B 0,C 180,E1 -10805.989,E2 -10805.989} C_VEL
LIN {X 0,Y 404.268,Z 236.624,A -85,B 0,C 180,E1 -10809.005,E2 -10809.005} C_VEL
LIN {X 0,Y 404.266,Z 236.625,A -85,B 0,C 180,E1 -10812.045,E2 -10812.045} C_VEL
LIN {X 0,Y 404.217,Z 236.632,A -85,B 0,C 180,E1 -10815.121,E2 -10815.121} C_VEL
LIN {X 0,Y 404.218,Z 236.631,A -85,B 0,C 180,E1 -10818.241,E2 -10818.241} C_VEL
LIN {X 0,Y 404.152,Z 236.639,A -85,B 0,C 180,E1 -10821.422,E2 -10821.422} C_VEL
LIN {X 0,Y 404.163,Z 236.64,A -85,B 0,C 180,E1 -10824.67,E2 -10824.67} C_VEL
LIN {X 0,Y 404.118,Z 236.642,A -85,B 0,C 180,E1 -10828.009,E2 -10828.009} C_VEL
LIN {X 0,Y 404.158,Z 236.637,A -85,B 0,C 180,E1 -10830.287,E2 -10830.287} C_VEL
LIN {X 0,Y 404.154,Z 236.639,A -85,B 0,C 180,E1 -10833.815,E2 -10833.815} C_VEL
LIN {X 0,Y 404.15,Z 236.64,A -85,B 0,C 180,E1 -10836.876,E2 -10836.876} C_VEL
LIN {X 0,Y 404.133,Z 236.641,A -85,B 0,C 180,E1 -10840.076,E2 -10840.076} C_VEL
LIN {X 0,Y 404.158,Z 236.639,A -85,B 0,C 180,E1 -10843.083,E2 -10843.083} C_VEL
LIN {X 0,Y 404.135,Z 236.644,A -85,B 0,C 180,E1 -10845.923,E2 -10845.923} C_VEL
LIN {X 0,Y 404.117,Z 236.642,A -85,B 0,C 180,E1 -10848.633,E2 -10848.633} C_VEL
LIN {X 0,Y 404.156,Z 236.64,A -85,B 0,C 180,E1 -10851.495,E2 -10851.495} C_VEL
LIN {X 0,Y 404.199,Z 236.631,A -85,B 0,C 180,E1 -10854.984,E2 -10854.984} C_VEL
LIN {X 0,Y 404.155,Z 236.643,A -85,B 0,C 180,E1 -10858.442,E2 -10858.442} C_VEL
LIN {X 0,Y 404.171,Z 236.64,A -85,B 0,C 180,E1 -10860.863,E2 -10860.863} C_VEL
LIN {X 0,Y 404.229,Z 236.764,A -85,B 0,C 180,E1 -10863.333,E2 -10863.333} C_VEL
LIN {X 0,Y 406.665,Z 249.438,A -85,B 0,C 180,E1 -10866.345,E2 -10866.345} C_VEL
LIN {X 0,Y 406.696,Z 254.173,A -85,B 0,C 180,E1 -10867.386,E2 -10867.386} C_VEL
LIN {X 0,Y 405.708,Z 269.101,A -85,B 0,C 180,E1 -10870.552,E2 -10870.552} C_VEL
LIN {X 0,Y 406.119,Z 272.315,A -85,B 0,C 180,E1 -10870.687,E2 -10870.687} C_VEL
LIN {X 0,Y 409.763,Z 296.104,A -85,B 0,C 180,E1 -10871.273,E2 -10871.273} C_VEL
LIN {X 0,Y 408.714,Z 376.597,A -85,B 0,C 180,E1 -10872.712,E2 -10872.712} C_VEL
LIN {X 0,Y 408.225,Z 389.99,A -85,B 0,C 180,E1 -10873.142,E2 -10873.142} C_VEL
LIN {X 0,Y 407.614,Z 403.372,A -85,B 0,C 180,E1 -10873.792,E2 -10873.792} C_VEL
LIN {X 0,Y 406.868,Z 415.383,A -85,B 0,C 180,E1 -10874.597,E2 -10874.597} C_VEL
LIN {X 0,Y 406.064,Z 427.514,A -85,B 0,C 180,E1 -10875.654,E2 -10875.654} C_VEL
LIN {X 0,Y 405.356,Z 437.252,A -85,B 0,C 180,E1 -10876.718,E2 -10876.718} C_VEL
LIN {X 0,Y 404.688,Z 446.542,A -85,B 0,C 180,E1 -10877.97,E2 -10877.97} C_VEL
LIN {X 0,Y 404.003,Z 455.558,A -85,B 0,C 180,E1 -10879.474,E2 -10879.474} C_VEL
LIN {X 0,Y 403.553,Z 462.812,A -85,B 0,C 180,E1 -10880.981,E2 -10880.981} C_VEL
LIN {X 0,Y 403.168,Z 468.583,A -85,B 0,C 180,E1 -10882.486,E2 -10882.486} C_VEL
LIN {X 0,Y 402.95,Z 473.119,A -85,B 0,C 180,E1 -10883.992,E2 -10883.992} C_VEL
LIN {X 0,Y 402.946,Z 475.508,A -85,B 0,C 180,E1 -10884.996,E2 -10884.996} C_VEL
LIN {X 0,Y 402.846,Z 477.461,A -85,B 0,C 180,E1 -10885.997,E2 -10885.997} C_VEL
LIN {X 0,Y 402.789,Z 478.997,A -85,B 0,C 180,E1 -10886.998,E2 -10886.998} C_VEL
LIN {X 0,Y 402.827,Z 480.081,A -85,B 0,C 180,E1 -10887.999,E2 -10887.999} C_VEL
LIN {X 0,Y 402.85,Z 480.762,A -85,B 0,C 180,E1 -10888.999,E2 -10888.999} C_VEL
LIN {X 0,Y 402.85,Z 480.963,A -85,B 0,C 180,E1 -10890.998,E2 -10890.998} C_VEL
LIN {X 0,Y 402.826,Z 480.44,A -85,B 0,C 180,E1 -10891.998,E2 -10891.998} C_VEL
LIN {X 0,Y 402.849,Z 478.2,A -85,B 0,C 180,E1 -10894,E2 -10894} C_VEL
LIN {X 0,Y 402.98,Z 475.421,A -85,B 0,C 180,E1 -10895.503,E2 -10895.503} C_VEL
LIN {X 0,Y 403.114,Z 471.627,A -85,B 0,C 180,E1 -10897.008,E2 -10897.008} C_VEL
LIN {X 0,Y 403.466,Z 466.72,A -85,B 0,C 180,E1 -10898.513,E2 -10898.513} C_VEL
LIN {X 0,Y 403.947,Z 460.555,A -85,B 0,C 180,E1 -10900.018,E2 -10900.018} C_VEL
LIN {X 0,Y 404.59,Z 452.893,A -85,B 0,C 180,E1 -10901.521,E2 -10901.521} C_VEL
LIN {X 0,Y 405.524,Z 443.284,A -85,B 0,C 180,E1 -10903.019,E2 -10903.019} C_VEL
LIN {X 0,Y 406.402,Z 433.607,A -85,B 0,C 180,E1 -10904.238,E2 -10904.238} C_VEL
LIN {X 0,Y 407.156,Z 423.659,A -85,B 0,C 180,E1 -10905.26,E2 -10905.26} C_VEL
LIN {X 0,Y 408.075,Z 411.371,A -85,B 0,C 180,E1 -10906.25,E2 -10906.25} C_VEL
LIN {X 0,Y 409.007,Z 399.346,A -85,B 0,C 180,E1 -10906.983,E2 -10906.983} C_VEL
LIN {X 0,Y 409.583,Z 387.028,A -85,B 0,C 180,E1 -10907.537,E2 -10907.537} C_VEL
LIN {X 0,Y 410.099,Z 374.335,A -85,B 0,C 180,E1 -10907.901,E2 -10907.901} C_VEL
LIN {X 0,Y 411.083,Z 294.87,A -85,B 0,C 180,E1 -10909.347,E2 -10909.347} C_VEL
LIN {X 0,Y 407.984,Z 277.076,A -85,B 0,C 180,E1 -10909.86,E2 -10909.86} C_VEL
LIN {X 0,Y 406.344,Z 268.943,A -85,B 0,C 180,E1 -10910.148,E2 -10910.148} C_VEL
LIN {X 0,Y 407.374,Z 255.066,A -85,B 0,C 180,E1 -10913.107,E2 -10913.107} C_VEL
LIN {X 0,Y 407.287,Z 251.764,A -85,B 0,C 180,E1 -10913.854,E2 -10913.854} C_VEL
LIN {X 0,Y 405.098,Z 240.718,A -85,B 0,C 180,E1 -10916.532,E2 -10916.532} C_VEL
LIN {X 0,Y 404.216,Z 236.69,A -85,B 0,C 180,E1 -10917.61,E2 -10917.61} C_VEL
LIN {X 0,Y 404.15,Z 236.641,A -85,B 0,C 180,E1 -10920.283,E2 -10920.283} C_VEL
LIN {X 0,Y 404.149,Z 236.645,A -85,B 0,C 180,E1 -10923.81,E2 -10923.81} C_VEL
LIN {X 0,Y 404.137,Z 236.643,A -85,B 0,C 180,E1 -10926.872,E2 -10926.872} C_VEL
LIN {X 0,Y 404.15,Z 236.645,A -85,B 0,C 180,E1 -10930.077,E2 -10930.077} C_VEL
LIN {X 0,Y 404.151,Z 236.638,A -85,B 0,C 180,E1 -10933.08,E2 -10933.08} C_VEL
LIN {X 0,Y 404.147,Z 236.634,A -85,B 0,C 180,E1 -10935.923,E2 -10935.923} C_VEL
LIN {X 0,Y 404.108,Z 236.649,A -85,B 0,C 180,E1 -10938.63,E2 -10938.63} C_VEL
LIN {X 0,Y 404.139,Z 236.64,A -85,B 0,C 180,E1 -10941.492,E2 -10941.492} C_VEL
LIN {X 0,Y 404.182,Z 236.638,A -85,B 0,C 180,E1 -10944.981,E2 -10944.981} C_VEL
LIN {X 0,Y 404.139,Z 236.644,A -85,B 0,C 180,E1 -10948.55,E2 -10948.55} C_VEL
LIN {X 0,Y 404.15,Z 236.639,A -85,B 0,C 180,E1 -10950.859,E2 -10950.859} C_VEL
LIN {X 0,Y 404.136,Z 236.641,A -85,B 0,C 180,E1 -10954.227,E2 -10954.227} C_VEL
LIN {X 0,Y 404.161,Z 236.637,A -85,B 0,C 180,E1 -10957.504,E2 -10957.504} C_VEL
LIN {X 0,Y 404.156,Z 236.64,A -85,B 0,C 180,E1 -10960.704,E2 -10960.704} C_VEL
LIN {X 0,Y 404.212,Z 236.628,A -85,B 0,C 180,E1 -10963.844,E2 -10963.844} C_VEL
LIN {X 0,Y 404.275,Z 236.625,A -85,B 0,C 180,E1 -10966.935,E2 -10966.935} C_VEL
LIN {X 0,Y 404.239,Z 236.629,A -85,B 0,C 180,E1 -10969.984,E2 -10969.984} C_VEL
LIN {X 0,Y 404.37,Z 236.607,A -85,B 0,C 180,E1 -10973.008,E2 -10973.008} C_VEL
LIN {X 0,Y 404.25,Z 236.629,A -85,B 0,C 180,E1 -10975.01,E2 -10975.01} C_VEL
LIN {X 0,Y 404.455,Z 236.602,A -85,B 0,C 180,E1 -10978.005,E2 -10978.005} C_VEL
LIN {X 0,Y 404.456,Z 236.602,A -85,B 0,C 180,E1 -10981.988,E2 -10981.988} C_VEL
LIN {X 0,Y 404.32,Z 236.616,A -85,B 0,C 180,E1 -10986.475,E2 -10986.475} C_VEL
LIN {X 0,Y 404.246,Z 236.625,A -85,B 0,C 180,E1 -10988.998,E2 -10988.998} C_VEL
LIN {X 0,Y 404.235,Z 236.631,A -85,B 0,C 180,E1 -10992.038,E2 -10992.038} C_VEL
LIN {X 0,Y 404.182,Z 236.636,A -85,B 0,C 180,E1 -10995.114,E2 -10995.114} C_VEL
LIN {X 0,Y 404.18,Z 236.64,A -85,B 0,C 180,E1 -10998.235,E2 -10998.235} C_VEL
LIN {X 0,Y 404.113,Z 236.645,A -85,B 0,C 180,E1 -11001.416,E2 -11001.416} C_VEL
LIN {X 0,Y 404.147,Z 236.64,A -85,B 0,C 180,E1 -11004.662,E2 -11004.662} C_VEL
LIN {X 0,Y 404.166,Z 236.634,A -85,B 0,C 180,E1 -11007.996,E2 -11007.996} C_VEL
LIN {X 0,Y 404.108,Z 236.645,A -85,B 0,C 180,E1 -11011.555,E2 -11011.555} C_VEL
LIN {X 0,Y 404.153,Z 236.637,A -85,B 0,C 180,E1 -11015.013,E2 -11015.013} C_VEL
LIN {X 0,Y 404.13,Z 236.643,A -85,B 0,C 180,E1 -11018.753,E2 -11018.753} C_VEL
LIN {X 0,Y 404.156,Z 236.643,A -85,B 0,C 180,E1 -11021.608,E2 -11021.608} C_VEL
LIN {X 0,Y 404.163,Z 236.721,A -85,B 0,C 180,E1 -11023.663,E2 -11023.663} C_VEL
LIN {X 0,Y 406.274,Z 246.74,A -85,B 0,C 180,E1 -11026.218,E2 -11026.218} C_VEL
LIN {X 0,Y 406.923,Z 251.57,A -85,B 0,C 180,E1 -11027.372,E2 -11027.372} C_VEL
LIN {X 0,Y 406.543,Z 258.767,A -85,B 0,C 180,E1 -11028.908,E2 -11028.908} C_VEL
LIN {X 0,Y 408.871,Z 269.34,A -85,B 0,C 180,E1 -11029.283,E2 -11029.283} C_VEL
LIN {X 0,Y 411.333,Z 282.953,A -85,B 0,C 180,E1 -11029.681,E2 -11029.681} C_VEL
LIN {X 0,Y 410.055,Z 366.292,A -85,B 0,C 180,E1 -11031.199,E2 -11031.199} C_VEL
LIN {X 0,Y 409.509,Z 379.897,A -85,B 0,C 180,E1 -11031.649,E2 -11031.649} C_VEL
LIN {X 0,Y 408.902,Z 391.818,A -85,B 0,C 180,E1 -11032.235,E2 -11032.235} C_VEL
LIN {X 0,Y 408.227,Z 402.725,A -85,B 0,C 180,E1 -11032.949,E2 -11032.949} C_VEL
LIN {X 0,Y 407.339,Z 414.359,A -85,B 0,C 180,E1 -11033.932,E2 -11033.932} C_VEL
LIN {X 0,Y 406.398,Z 424.906,A -85,B 0,C 180,E1 -11035.054,E2 -11035.054} C_VEL
LIN {X 0,Y 405.543,Z 434.53,A -85,B 0,C 180,E1 -11036.322,E2 -11036.322} C_VEL
LIN {X 0,Y 404.766,Z 442.954,A -85,B 0,C 180,E1 -11037.699,E2 -11037.699} C_VEL
LIN {X 0,Y 404.142,Z 450.106,A -85,B 0,C 180,E1 -11039.138,E2 -11039.138} C_VEL
LIN {X 0,Y 403.639,Z 456.784,A -85,B 0,C 180,E1 -11040.824,E2 -11040.824} C_VEL
LIN {X 0,Y 403.275,Z 461.576,A -85,B 0,C 180,E1 -11042.38,E2 -11042.38} C_VEL
LIN {X 0,Y 402.977,Z 465.614,A -85,B 0,C 180,E1 -11044.153,E2 -11044.153} C_VEL
LIN {X 0,Y 402.796,Z 467.407,A -85,B 0,C 180,E1 -11045.246,E2 -11045.246} C_VEL
LIN {X 0,Y 402.668,Z 468.735,A -85,B 0,C 180,E1 -11046.334,E2 -11046.334} C_VEL
LIN {X 0,Y 402.613,Z 469.665,A -85,B 0,C 180,E1 -11047.678,E2 -11047.678} C_VEL
LIN {X 0,Y 402.613,Z 469.817,A -85,B 0,C 180,E1 -11049.568,E2 -11049.568} C_VEL
LIN {X 0,Y 402.689,Z 469.247,A -85,B 0,C 180,E1 -11050.636,E2 -11050.636} C_VEL
LIN {X 0,Y 402.677,Z 468.245,A -85,B 0,C 180,E1 -11051.692,E2 -11051.692} C_VEL
LIN {X 0,Y 402.88,Z 465.291,A -85,B 0,C 180,E1 -11053.604,E2 -11053.604} C_VEL
LIN {X 0,Y 403.115,Z 461.113,A -85,B 0,C 180,E1 -11055.359,E2 -11055.359} C_VEL
LIN {X 0,Y 403.405,Z 456.168,A -85,B 0,C 180,E1 -11056.912,E2 -11056.912} C_VEL
LIN {X 0,Y 403.816,Z 449.911,A -85,B 0,C 180,E1 -11058.456,E2 -11058.456} C_VEL
LIN {X 0,Y 404.329,Z 442.132,A -85,B 0,C 180,E1 -11059.992,E2 -11059.992} C_VEL
LIN {X 0,Y 405.077,Z 432.957,A -85,B 0,C 180,E1 -11061.429,E2 -11061.429} C_VEL
LIN {X 0,Y 405.758,Z 423.243,A -85,B 0,C 180,E1 -11062.663,E2 -11062.663} C_VEL
LIN {X 0,Y 406.539,Z 413.408,A -85,B 0,C 180,E1 -11063.674,E2 -11063.674} C_VEL
LIN {X 0,Y 407.185,Z 402.845,A -85,B 0,C 180,E1 -11064.554,E2 -11064.554} C_VEL
LIN {X 0,Y 407.819,Z 390.134,A -85,B 0,C 180,E1 -11065.368,E2 -11065.368} C_VEL
LIN {X 0,Y 408.41,Z 377.337,A -85,B 0,C 180,E1 -11065.962,E2 -11065.962} C_VEL
LIN {X 0,Y 408.733,Z 367.626,A -85,B 0,C 180,E1 -11066.272,E2 -11066.272} C_VEL
LIN {X 0,Y 408.177,Z 361.862,A -85,B 0,C 180,E1 -11066.439,E2 -11066.439} C_VEL
LIN {X 0,Y 402.84,Z 343.155,A -85,B 0,C 180,E1 -11066.991,E2 -11066.991} C_VEL
LIN {X 0,Y 402.29,Z 337.338,A -85,B 0,C 180,E1 -11067.116,E2 -11067.116} C_VEL
LIN {X 0,Y 402.896,Z 281.534,A -85,B 0,C 180,E1 -11068.128,E2 -11068.128} C_VEL
LIN {X 0,Y 398.993,Z 259.307,A -85,B 0,C 180,E1 -11068.74,E2 -11068.74} C_VEL
LIN {X 0,Y 399.002,Z 257.737,A -85,B 0,C 180,E1 -11068.992,E2 -11068.992} C_VEL
LIN {X 0,Y 399.446,Z 249.118,A -85,B 0,C 180,E1 -11071.01,E2 -11071.01} C_VEL
LIN {X 0,Y 397.678,Z 239.972,A -85,B 0,C 180,E1 -11073.294,E2 -11073.294} C_VEL
LIN {X 0,Y 397.128,Z 237.548,A -85,B 0,C 180,E1 -11073.997,E2 -11073.997} C_VEL
LIN {X 0,Y 397.33,Z 237.493,A -85,B 0,C 180,E1 -11076.094,E2 -11076.094} C_VEL
LIN {X 0,Y 397.213,Z 237.505,A -85,B 0,C 180,E1 -11079.164,E2 -11079.164} C_VEL
LIN {X 0,Y 397.189,Z 237.506,A -85,B 0,C 180,E1 -11082.261,E2 -11082.261} C_VEL
LIN {X 0,Y 397.141,Z 237.514,A -85,B 0,C 180,E1 -11085.395,E2 -11085.395} C_VEL
LIN {X 0,Y 397.124,Z 237.513,A -85,B 0,C 180,E1 -11088.577,E2 -11088.577} C_VEL
LIN {X 0,Y 397.059,Z 237.527,A -85,B 0,C 180,E1 -11091.822,E2 -11091.822} C_VEL
LIN {X 0,Y 397.073,Z 237.519,A -85,B 0,C 180,E1 -11095.139,E2 -11095.139} C_VEL
LIN {X 0,Y 397.045,Z 237.526,A -85,B 0,C 180,E1 -11098.551,E2 -11098.551} C_VEL
LIN {X 0,Y 397.05,Z 237.525,A -85,B 0,C 180,E1 -11101.84,E2 -11101.84} C_VEL
LIN {X 0,Y 397.087,Z 237.523,A -85,B 0,C 180,E1 -11104.499,E2 -11104.499} C_VEL
LIN {X 0,Y 397.062,Z 237.526,A -85,B 0,C 180,E1 -11108.281,E2 -11108.281} C_VEL
LIN {X 0,Y 397.027,Z 237.526,A -85,B 0,C 180,E1 -11111.981,E2 -11111.981} C_VEL
LIN {X 0,Y 397.063,Z 237.524,A -85,B 0,C 180,E1 -11115.074,E2 -11115.074} C_VEL
LIN {X 0,Y 397.033,Z 237.525,A -85,B 0,C 180,E1 -11118.028,E2 -11118.028} C_VEL
LIN {X 0,Y 397.075,Z 237.519,A -85,B 0,C 180,E1 -11121.729,E2 -11121.729} C_VEL
LIN {X 0,Y 397.103,Z 237.518,A -85,B 0,C 180,E1 -11125.511,E2 -11125.511} C_VEL
LIN {X 0,Y 397.064,Z 237.528,A -85,B 0,C 180,E1 -11129.122,E2 -11129.122} C_VEL
LIN {X 0,Y 397.051,Z 237.522,A -85,B 0,C 180,E1 -11132.257,E2 -11132.257} C_VEL
LIN {X 0,Y 397.094,Z 237.519,A -85,B 0,C 180,E1 -11134.87,E2 -11134.87} C_VEL
LIN {X 0,Y 397.089,Z 237.518,A -85,B 0,C 180,E1 -11138.186,E2 -11138.186} C_VEL
LIN {X 0,Y 397.153,Z 237.515,A -85,B 0,C 180,E1 -11141.431,E2 -11141.431} C_VEL
LIN {X 0,Y 397.174,Z 237.507,A -85,B 0,C 180,E1 -11144.612,E2 -11144.612} C_VEL
LIN {X 0,Y 397.214,Z 237.509,A -85,B 0,C 180,E1 -11147.746,E2 -11147.746} C_VEL
LIN {X 0,Y 397.23,Z 237.5,A -85,B 0,C 180,E1 -11150.842,E2 -11150.842} C_VEL
LIN {X 0,Y 397.323,Z 237.495,A -85,B 0,C 180,E1 -11153.912,E2 -11153.912} C_VEL
LIN {X 0,Y 397.446,Z 237.479,A -85,B 0,C 180,E1 -11157.977,E2 -11157.977} C_VEL
LIN {X 0,Y 397.444,Z 237.478,A -85,B 0,C 180,E1 -11162.031,E2 -11162.031} C_VEL
LIN {X 0,Y 397.329,Z 237.492,A -85,B 0,C 180,E1 -11166.096,E2 -11166.096} C_VEL
LIN {X 0,Y 397.24,Z 237.499,A -85,B 0,C 180,E1 -11169.166,E2 -11169.166} C_VEL
LIN {X 0,Y 397.23,Z 237.504,A -85,B 0,C 180,E1 -11172.261,E2 -11172.261} C_VEL
LIN {X 0,Y 397.19,Z 237.505,A -85,B 0,C 180,E1 -11175.395,E2 -11175.395} C_VEL
LIN {X 0,Y 397.171,Z 237.512,A -85,B 0,C 180,E1 -11178.576,E2 -11178.576} C_VEL
LIN {X 0,Y 397.109,Z 237.515,A -85,B 0,C 180,E1 -11181.821,E2 -11181.821} C_VEL
LIN {X 0,Y 397.111,Z 237.52,A -85,B 0,C 180,E1 -11185.138,E2 -11185.138} C_VEL
LIN {X 0,Y 397.078,Z 237.52,A -85,B 0,C 180,E1 -11188.55,E2 -11188.55} C_VEL
LIN {X 0,Y 397.095,Z 237.517,A -85,B 0,C 180,E1 -11191.837,E2 -11191.837} C_VEL
LIN {X 0,Y 397.135,Z 237.512,A -85,B 0,C 180,E1 -11194.496,E2 -11194.496} C_VEL
LIN {X 0,Y 397.108,Z 237.515,A -85,B 0,C 180,E1 -11198.278,E2 -11198.278} C_VEL
LIN {X 0,Y 397.067,Z 237.522,A -85,B 0,C 180,E1 -11201.977,E2 -11201.977} C_VEL
LIN {X 0,Y 397.1,Z 237.517,A -85,B 0,C 180,E1 -11205.07,E2 -11205.07} C_VEL
LIN {X 0,Y 397.067,Z 237.524,A -85,B 0,C 180,E1 -11208.024,E2 -11208.024} C_VEL
LIN {X 0,Y 397.108,Z 237.521,A -85,B 0,C 180,E1 -11211.724,E2 -11211.724} C_VEL
LIN {X 0,Y 397.141,Z 237.513,A -85,B 0,C 180,E1 -11215.507,E2 -11215.507} C_VEL
LIN {X 0,Y 397.093,Z 237.52,A -85,B 0,C 180,E1 -11219.117,E2 -11219.117} C_VEL
LIN {X 0,Y 397.141,Z 237.516,A -85,B 0,C 180,E1 -11222.604,E2 -11222.604} C_VEL
LIN {X 0,Y 397.173,Z 237.637,A -85,B 0,C 180,E1 -11223.105,E2 -11223.105} C_VEL
LIN {X 0,Y 399.599,Z 250.221,A -85,B 0,C 180,E1 -11226.147,E2 -11226.147} C_VEL
LIN {X 0,Y 399.839,Z 253.864,A -85,B 0,C 180,E1 -11226.976,E2 -11226.976} C_VEL
LIN {X 0,Y 398.766,Z 268.894,A -85,B 0,C 180,E1 -11230.233,E2 -11230.233} C_VEL
LIN {X 0,Y 399.046,Z 271.385,A -85,B 0,C 180,E1 -11230.365,E2 -11230.365} C_VEL
LIN {X 0,Y 402.946,Z 296.159,A -85,B 0,C 180,E1 -11230.994,E2 -11230.994} C_VEL
LIN {X 0,Y 401.848,Z 377.169,A -85,B 0,C 180,E1 -11232.472,E2 -11232.472} C_VEL
LIN {X 0,Y 401.318,Z 391.092,A -85,B 0,C 180,E1 -11232.941,E2 -11232.941} C_VEL
LIN {X 0,Y 400.696,Z 403.58,A -85,B 0,C 180,E1 -11233.57,E2 -11233.57} C_VEL
LIN {X 0,Y 399.963,Z 414.713,A -85,B 0,C 180,E1 -11234.325,E2 -11234.325} C_VEL
LIN {X 0,Y 399.135,Z 426.829,A -85,B 0,C 180,E1 -11235.387,E2 -11235.387} C_VEL
LIN {X 0,Y 398.428,Z 436.933,A -85,B 0,C 180,E1 -11236.501,E2 -11236.501} C_VEL
LIN {X 0,Y 397.714,Z 446.151,A -85,B 0,C 180,E1 -11237.756,E2 -11237.756} C_VEL
LIN {X 0,Y 396.984,Z 455.217,A -85,B 0,C 180,E1 -11239.286,E2 -11239.286} C_VEL
LIN {X 0,Y 396.492,Z 462.515,A -85,B 0,C 180,E1 -11240.819,E2 -11240.819} C_VEL
LIN {X 0,Y 396.097,Z 468.339,A -85,B 0,C 180,E1 -11242.351,E2 -11242.351} C_VEL
LIN {X 0,Y 395.844,Z 473.654,A -85,B 0,C 180,E1 -11244.185,E2 -11244.185} C_VEL
LIN {X 0,Y 395.771,Z 477.29,A -85,B 0,C 180,E1 -11245.925,E2 -11245.925} C_VEL
LIN {X 0,Y 395.695,Z 478.843,A -85,B 0,C 180,E1 -11246.944,E2 -11246.944} C_VEL
LIN {X 0,Y 395.724,Z 479.95,A -85,B 0,C 180,E1 -11247.963,E2 -11247.963} C_VEL
LIN {X 0,Y 395.761,Z 480.644,A -85,B 0,C 180,E1 -11248.981,E2 -11248.981} C_VEL
LIN {X 0,Y 395.765,Z 480.951,A -85,B 0,C 180,E1 -11249.998,E2 -11249.998} C_VEL
LIN {X 0,Y 395.761,Z 480.873,A -85,B 0,C 180,E1 -11251.016,E2 -11251.016} C_VEL
LIN {X 0,Y 395.723,Z 480.374,A -85,B 0,C 180,E1 -11252.034,E2 -11252.034} C_VEL
LIN {X 0,Y 395.775,Z 478.163,A -85,B 0,C 180,E1 -11254.072,E2 -11254.072} C_VEL
LIN {X 0,Y 395.885,Z 475.412,A -85,B 0,C 180,E1 -11255.602,E2 -11255.602} C_VEL
LIN {X 0,Y 396.064,Z 471.647,A -85,B 0,C 180,E1 -11257.134,E2 -11257.134} C_VEL
LIN {X 0,Y 396.417,Z 466.772,A -85,B 0,C 180,E1 -11258.666,E2 -11258.666} C_VEL
LIN {X 0,Y 396.942,Z 460.641,A -85,B 0,C 180,E1 -11260.196,E2 -11260.196} C_VEL
LIN {X 0,Y 397.635,Z 453.03,A -85,B 0,C 180,E1 -11261.726,E2 -11261.726} C_VEL
LIN {X 0,Y 398.612,Z 443.478,A -85,B 0,C 180,E1 -11263.249,E2 -11263.249} C_VEL
LIN {X 0,Y 399.537,Z 433.258,A -85,B 0,C 180,E1 -11264.562,E2 -11264.562} C_VEL
LIN {X 0,Y 400.462,Z 422.621,A -85,B 0,C 180,E1 -11265.652,E2 -11265.652} C_VEL
LIN {X 0,Y 401.305,Z 411.848,A -85,B 0,C 180,E1 -11266.532,E2 -11266.532} C_VEL
LIN {X 0,Y 402.303,Z 398.866,A -85,B 0,C 180,E1 -11267.34,E2 -11267.34} C_VEL
LIN {X 0,Y 402.936,Z 386.316,A -85,B 0,C 180,E1 -11267.902,E2 -11267.902} C_VEL
LIN {X 0,Y 403.46,Z 373.244,A -85,B 0,C 180,E1 -11268.271,E2 -11268.271} C_VEL
LIN {X 0,Y 404.508,Z 295.974,A -85,B 0,C 180,E1 -11269.697,E2 -11269.697} C_VEL
LIN {X 0,Y 401.762,Z 279.838,A -85,B 0,C 180,E1 -11270.17,E2 -11270.17} C_VEL
LIN {X 0,Y 399.523,Z 268.895,A -85,B 0,C 180,E1 -11270.556,E2 -11270.556} C_VEL
LIN {X 0,Y 400.56,Z 255.216,A -85,B 0,C 180,E1 -11273.524,E2 -11273.524} C_VEL
LIN {X 0,Y 399.438,Z 248.133,A -85,B 0,C 180,E1 -11275.235,E2 -11275.235} C_VEL
LIN {X 0,Y 397.2,Z 237.778,A -85,B 0,C 180,E1 -11277.884,E2 -11277.884} C_VEL
LIN {X 0,Y 397.126,Z 237.517,A -85,B 0,C 180,E1 -11278.541,E2 -11278.541} C_VEL
LIN {X 0,Y 397.082,Z 237.521,A -85,B 0,C 180,E1 -11282.069,E2 -11282.069} C_VEL
LIN {X 0,Y 397.122,Z 237.512,A -85,B 0,C 180,E1 -11285.5,E2 -11285.5} C_VEL
LIN {X 0,Y 397.104,Z 237.515,A -85,B 0,C 180,E1 -11288.853,E2 -11288.853} C_VEL
LIN {X 0,Y 397.065,Z 237.516,A -85,B 0,C 180,E1 -11292.265,E2 -11292.265} C_VEL
LIN {X 0,Y 397.086,Z 237.518,A -85,B 0,C 180,E1 -11295.066,E2 -11295.066} C_VEL
LIN {X 0,Y 397.058,Z 237.518,A -85,B 0,C 180,E1 -11298.02,E2 -11298.02} C_VEL
LIN {X 0,Y 397.091,Z 237.518,A -85,B 0,C 180,E1 -11301.72,E2 -11301.72} C_VEL
LIN {X 0,Y 397.123,Z 237.515,A -85,B 0,C 180,E1 -11305.503,E2 -11305.503} C_VEL
LIN {X 0,Y 397.075,Z 237.523,A -85,B 0,C 180,E1 -11309.114,E2 -11309.114} C_VEL
LIN {X 0,Y 397.09,Z 237.523,A -85,B 0,C 180,E1 -11312.599,E2 -11312.599} C_VEL
LIN {X 0,Y 397.107,Z 237.515,A -85,B 0,C 180,E1 -11315.977,E2 -11315.977} C_VEL
LIN {X 0,Y 397.133,Z 237.511,A -85,B 0,C 180,E1 -11319.701,E2 -11319.701} C_VEL
LIN {X 0,Y 397.175,Z 237.507,A -85,B 0,C 180,E1 -11322.841,E2 -11322.841} C_VEL
LIN {X 0,Y 397.221,Z 237.504,A -85,B 0,C 180,E1 -11326.699,E2 -11326.699} C_VEL
LIN {X 0,Y 397.2,Z 237.507,A -85,B 0,C 180,E1 -11329.805,E2 -11329.805} C_VEL
LIN {X 0,Y 397.318,Z 237.484,A -85,B 0,C 180,E1 -11332.884,E2 -11332.884} C_VEL
LIN {X 0,Y 397.222,Z 237.504,A -85,B 0,C 180,E1 -11334.921,E2 -11334.921} C_VEL
LIN {X 0,Y 397.422,Z 237.479,A -85,B 0,C 180,E1 -11337.969,E2 -11337.969} C_VEL
LIN {X 0,Y 397.425,Z 237.478,A -85,B 0,C 180,E1 -11342.023,E2 -11342.023} C_VEL
LIN {X 0,Y 397.276,Z 237.494,A -85,B 0,C 180,E1 -11346.469,E2 -11346.469} C_VEL
LIN {X 0,Y 397.216,Z 237.502,A -85,B 0,C 180,E1 -11349.158,E2 -11349.158} C_VEL
LIN {X 0,Y 397.198,Z 237.505,A -85,B 0,C 180,E1 -11352.254,E2 -11352.254} C_VEL
LIN {X 0,Y 397.155,Z 237.513,A -85,B 0,C 180,E1 -11355.388,E2 -11355.388} C_VEL
LIN {X 0,Y 397.133,Z 237.515,A -85,B 0,C 180,E1 -11358.57,E2 -11358.57} C_VEL
LIN {X 0,Y 397.07,Z 237.526,A -85,B 0,C 180,E1 -11361.815,E2 -11361.815} C_VEL
LIN {X 0,Y 397.125,Z 237.512,A -85,B 0,C 180,E1 -11365.509,E2 -11365.509} C_VEL
LIN {X 0,Y 397.092,Z 237.511,A -85,B 0,C 180,E1 -11368.54,E2 -11368.54} C_VEL
LIN {X 0,Y 397.047,Z 237.522,A -85,B 0,C 180,E1 -11372.068,E2 -11372.068} C_VEL
LIN {X 0,Y 397.088,Z 237.515,A -85,B 0,C 180,E1 -11375.5,E2 -11375.5} C_VEL
LIN {X 0,Y 397.104,Z 237.519,A -85,B 0,C 180,E1 -11378.86,E2 -11378.86} C_VEL
LIN {X 0,Y 397.123,Z 237.517,A -85,B 0,C 180,E1 -11382.253,E2 -11382.253} C_VEL
LIN {X 0,Y 397.115,Z 237.596,A -85,B 0,C 180,E1 -11383.299,E2 -11383.299} C_VEL
LIN {X 0,Y 399.212,Z 247.404,A -85,B 0,C 180,E1 -11385.861,E2 -11385.861} C_VEL
LIN {X 0,Y 400.053,Z 252.958,A -85,B 0,C 180,E1 -11387.221,E2 -11387.221} C_VEL
LIN {X 0,Y 399.743,Z 258.916,A -85,B 0,C 180,E1 -11388.5,E2 -11388.5} C_VEL
LIN {X 0,Y 403.705,Z 277.446,A -85,B 0,C 180,E1 -11389.139,E2 -11389.139} C_VEL
LIN {X 0,Y 404.716,Z 282.837,A -85,B 0,C 180,E1 -11389.302,E2 -11389.302} C_VEL
LIN {X 0,Y 403.393,Z 366.626,A -85,B 0,C 180,E1 -11390.858,E2 -11390.858} C_VEL
LIN {X 0,Y 402.819,Z 380.289,A -85,B 0,C 180,E1 -11391.32,E2 -11391.32} C_VEL
LIN {X 0,Y 402.156,Z 392.843,A -85,B 0,C 180,E1 -11391.956,E2 -11391.956} C_VEL
LIN {X 0,Y 401.298,Z 405.389,A -85,B 0,C 180,E1 -11392.831,E2 -11392.831} C_VEL
LIN {X 0,Y 400.348,Z 416.676,A -85,B 0,C 180,E1 -11393.844,E2 -11393.844} C_VEL
LIN {X 0,Y 399.439,Z 426.696,A -85,B 0,C 180,E1 -11394.971,E2 -11394.971} C_VEL
LIN {X 0,Y 398.513,Z 436.084,A -85,B 0,C 180,E1 -11396.281,E2 -11396.281} C_VEL
LIN {X 0,Y 397.713,Z 444.288,A -85,B 0,C 180,E1 -11397.689,E2 -11397.689} C_VEL
LIN {X 0,Y 397.087,Z 451.082,A -85,B 0,C 180,E1 -11399.12,E2 -11399.12} C_VEL
LIN {X 0,Y 396.565,Z 457.575,A -85,B 0,C 180,E1 -11400.835,E2 -11400.835} C_VEL
LIN {X 0,Y 396.148,Z 462.477,A -85,B 0,C 180,E1 -11402.533,E2 -11402.533} C_VEL
LIN {X 0,Y 395.937,Z 465.006,A -85,B 0,C 180,E1 -11403.658,E2 -11403.658} C_VEL
LIN {X 0,Y 395.758,Z 467.175,A -85,B 0,C 180,E1 -11404.9,E2 -11404.9} C_VEL
LIN {X 0,Y 395.613,Z 468.444,A -85,B 0,C 180,E1 -11405.886,E2 -11405.886} C_VEL
LIN {X 0,Y 395.532,Z 469.712,A -85,B 0,C 180,E1 -11407.496,E2 -11407.496} C_VEL
LIN {X 0,Y 395.493,Z 469.975,A -85,B 0,C 180,E1 -11409.184,E2 -11409.184} C_VEL
LIN {X 0,Y 395.562,Z 469.561,A -85,B 0,C 180,E1 -11410.314,E2 -11410.314} C_VEL
LIN {X 0,Y 395.572,Z 468.725,A -85,B 0,C 180,E1 -11411.351,E2 -11411.351} C_VEL
LIN {X 0,Y 395.631,Z 467.407,A -85,B 0,C 180,E1 -11412.425,E2 -11412.425} C_VEL
LIN {X 0,Y 395.845,Z 464.583,A -85,B 0,C 180,E1 -11414.028,E2 -11414.028} C_VEL
LIN {X 0,Y 396.074,Z 460.677,A -85,B 0,C 180,E1 -11415.618,E2 -11415.618} C_VEL
LIN {X 0,Y 396.379,Z 455.097,A -85,B 0,C 180,E1 -11417.336,E2 -11417.336} C_VEL
LIN {X 0,Y 396.888,Z 447.948,A -85,B 0,C 180,E1 -11419.028,E2 -11419.028} C_VEL
LIN {X 0,Y 397.535,Z 439.611,A -85,B 0,C 180,E1 -11420.59,E2 -11420.59} C_VEL
LIN {X 0,Y 398.227,Z 431.075,A -85,B 0,C 180,E1 -11421.885,E2 -11421.885} C_VEL
LIN {X 0,Y 398.945,Z 421.723,A -85,B 0,C 180,E1 -11423.045,E2 -11423.045} C_VEL
LIN {X 0,Y 399.757,Z 411.469,A -85,B 0,C 180,E1 -11424.073,E2 -11424.073} C_VEL
LIN {X 0,Y 400.457,Z 400.341,A -85,B 0,C 180,E1 -11424.967,E2 -11424.967} C_VEL
LIN {X 0,Y 401.095,Z 388.02,A -85,B 0,C 180,E1 -11425.731,E2 -11425.731} C_VEL
LIN {X 0,Y 401.613,Z 375.374,A -85,B 0,C 180,E1 -11426.29,E2 -11426.29} C_VEL
LIN {X 0,Y 401.973,Z 361.858,A -85,B 0,C 180,E1 -11426.667,E2 -11426.667} C_VEL
LIN {X 0,Y 402.29,Z 337.338,A -85,B 0,C 180,E1 -11427.116,E2 -11427.116} C_VEL
LIN {X 0,Y 401.756,Z 331.529,A -85,B 0,C 180,E1 -11427.245,E2 -11427.245} C_VEL
LIN {X 0,Y 396.478,Z 312.816,A -85,B 0,C 180,E1 -11427.815,E2 -11427.815} C_VEL
LIN {X 0,Y 395.855,Z 307.008,A -85,B 0,C 180,E1 -11427.952,E2 -11427.952} C_VEL
LIN {X 0,Y 396.052,Z 282.048,A -85,B 0,C 180,E1 -11428.417,E2 -11428.417} C_VEL
LIN {X 0,Y 392.098,Z 259.486,A -85,B 0,C 180,E1 -11429.039,E2 -11429.039} C_VEL
LIN {X 0,Y 392.052,Z 258.183,A -85,B 0,C 180,E1 -11429.231,E2 -11429.231} C_VEL
LIN {X 0,Y 392.496,Z 250.565,A -85,B 0,C 180,E1 -11431.028,E2 -11431.028} C_VEL
LIN {X 0,Y 390.731,Z 241.417,A -85,B 0,C 180,E1 -11433.353,E2 -11433.353} C_VEL
LIN {X 0,Y 390.097,Z 238.418,A -85,B 0,C 180,E1 -11434.231,E2 -11434.231} C_VEL
LIN {X 0,Y 390.284,Z 238.37,A -85,B 0,C 180,E1 -11436.204,E2 -11436.204} C_VEL
LIN {X 0,Y 390.166,Z 238.385,A -85,B 0,C 180,E1 -11439.331,E2 -11439.331} C_VEL
LIN {X 0,Y 390.138,Z 238.383,A -85,B 0,C 180,E1 -11442.486,E2 -11442.486} C_VEL
LIN {X 0,Y 390.101,Z 238.395,A -85,B 0,C 180,E1 -11445.68,E2 -11445.68} C_VEL
LIN {X 0,Y 390.068,Z 238.392,A -85,B 0,C 180,E1 -11448.925,E2 -11448.925} C_VEL
LIN {X 0,Y 390.001,Z 238.404,A -85,B 0,C 180,E1 -11452.238,E2 -11452.238} C_VEL
LIN {X 0,Y 390.017,Z 238.402,A -85,B 0,C 180,E1 -11455.726,E2 -11455.726} C_VEL
LIN {X 0,Y 390,Z 238.4,A -85,B 0,C 180,E1 -11459.116,E2 -11459.116} C_VEL
LIN {X 0,Y 390.011,Z 238.401,A -85,B 0,C 180,E1 -11462.726,E2 -11462.726} C_VEL
LIN {X 0,Y 390.013,Z 238.4,A -85,B 0,C 180,E1 -11465.827,E2 -11465.827} C_VEL
LIN {X 0,Y 390.009,Z 238.4,A -85,B 0,C 180,E1 -11469.216,E2 -11469.216} C_VEL
LIN {X 0,Y 390.006,Z 238.404,A -85,B 0,C 180,E1 -11472.377,E2 -11472.377} C_VEL
LIN {X 0,Y 390.02,Z 238.399,A -85,B 0,C 180,E1 -11475.359,E2 -11475.359} C_VEL
LIN {X 0,Y 389.996,Z 238.402,A -85,B 0,C 180,E1 -11478.19,E2 -11478.19} C_VEL
LIN {X 0,Y 390.04,Z 238.403,A -85,B 0,C 180,E1 -11480.909,E2 -11480.909} C_VEL
LIN {X 0,Y 390.054,Z 238.398,A -85,B 0,C 180,E1 -11484.796,E2 -11484.796} C_VEL
LIN {X 0,Y 390.008,Z 238.4,A -85,B 0,C 180,E1 -11488.5,E2 -11488.5} C_VEL
LIN {X 0,Y 390.005,Z 238.4,A -85,B 0,C 180,E1 -11492.008,E2 -11492.008} C_VEL
LIN {X 0,Y 390.035,Z 238.402,A -85,B 0,C 180,E1 -11495.522,E2 -11495.522} C_VEL
LIN {X 0,Y 390.05,Z 238.395,A -85,B 0,C 180,E1 -11498.883,E2 -11498.883} C_VEL
LIN {X 0,Y 390.108,Z 238.388,A -85,B 0,C 180,E1 -11502.171,E2 -11502.171} C_VEL
LIN {X 0,Y 390.141,Z 238.387,A -85,B 0,C 180,E1 -11505.397,E2 -11505.397} C_VEL
LIN {X 0,Y 390.138,Z 238.383,A -85,B 0,C 180,E1 -11508.575,E2 -11508.575} C_VEL
LIN {X 0,Y 390.259,Z 238.373,A -85,B 0,C 180,E1 -11512.091,E2 -11512.091} C_VEL
LIN {X 0,Y 390.203,Z 238.375,A -85,B 0,C 180,E1 -11514.837,E2 -11514.837} C_VEL
LIN {X 0,Y 390.413,Z 238.355,A -85,B 0,C 180,E1 -11517.941,E2 -11517.941} C_VEL
LIN {X 0,Y 390.411,Z 238.355,A -85,B 0,C 180,E1 -11522.067,E2 -11522.067} C_VEL
LIN {X 0,Y 390.285,Z 238.37,A -85,B 0,C 180,E1 -11526.206,E2 -11526.206} C_VEL
LIN {X 0,Y 390.198,Z 238.376,A -85,B 0,C 180,E1 -11529.333,E2 -11529.333} C_VEL
LIN {X 0,Y 390.182,Z 238.384,A -85,B 0,C 180,E1 -11532.486,E2 -11532.486} C_VEL
LIN {X 0,Y 390.151,Z 238.381,A -85,B 0,C 180,E1 -11535.68,E2 -11535.68} C_VEL
LIN {X 0,Y 390.116,Z 238.391,A -85,B 0,C 180,E1 -11538.925,E2 -11538.925} C_VEL
LIN {X 0,Y 390.049,Z 238.395,A -85,B 0,C 180,E1 -11542.237,E2 -11542.237} C_VEL
LIN {X 0,Y 390.065,Z 238.393,A -85,B 0,C 180,E1 -11545.724,E2 -11545.724} C_VEL
LIN {X 0,Y 390.04,Z 238.403,A -85,B 0,C 180,E1 -11549.114,E2 -11549.114} C_VEL
LIN {X 0,Y 390.057,Z 238.395,A -85,B 0,C 180,E1 -11552.723,E2 -11552.723} C_VEL
LIN {X 0,Y 390.069,Z 238.394,A -85,B 0,C 180,E1 -11555.826,E2 -11555.826} C_VEL
LIN {X 0,Y 390.053,Z 238.398,A -85,B 0,C 180,E1 -11559.213,E2 -11559.213} C_VEL
LIN {X 0,Y 390.046,Z 238.395,A -85,B 0,C 180,E1 -11562.373,E2 -11562.373} C_VEL
LIN {X 0,Y 390.056,Z 238.397,A -85,B 0,C 180,E1 -11565.354,E2 -11565.354} C_VEL
LIN {X 0,Y 390.03,Z 238.399,A -85,B 0,C 180,E1 -11568.185,E2 -11568.185} C_VEL
LIN {X 0,Y 390.074,Z 238.391,A -85,B 0,C 180,E1 -11570.904,E2 -11570.904} C_VEL
LIN {X 0,Y 390.101,Z 238.388,A -85,B 0,C 180,E1 -11574.793,E2 -11574.793} C_VEL
LIN {X 0,Y 390.039,Z 238.401,A -85,B 0,C 180,E1 -11578.495,E2 -11578.495} C_VEL
LIN {X 0,Y 390.053,Z 238.398,A -85,B 0,C 180,E1 -11582.063,E2 -11582.063} C_VEL
LIN {X 0,Y 390.122,Z 238.511,A -85,B 0,C 180,E1 -11582.869,E2 -11582.869} C_VEL
LIN {X 0,Y 392.354,Z 249.843,A -85,B 0,C 180,E1 -11585.669,E2 -11585.669} C_VEL
LIN {X 0,Y 392.889,Z 254.766,A -85,B 0,C 180,E1 -11586.824,E2 -11586.824} C_VEL
LIN {X 0,Y 391.853,Z 268.937,A -85,B 0,C 180,E1 -11589.938,E2 -11589.938} C_VEL
LIN {X 0,Y 392.432,Z 273.294,A -85,B 0,C 180,E1 -11590.105,E2 -11590.105} C_VEL
LIN {X 0,Y 396.136,Z 297.635,A -85,B 0,C 180,E1 -11590.732,E2 -11590.732} C_VEL
LIN {X 0,Y 395.01,Z 376.576,A -85,B 0,C 180,E1 -11592.192,E2 -11592.192} C_VEL
LIN {X 0,Y 394.491,Z 389.9,A -85,B 0,C 180,E1 -11592.637,E2 -11592.637} C_VEL
LIN {X 0,Y 393.83,Z 402.684,A -85,B 0,C 180,E1 -11593.275,E2 -11593.275} C_VEL
LIN {X 0,Y 393.113,Z 414.044,A -85,B 0,C 180,E1 -11594.044,E2 -11594.044} C_VEL
LIN {X 0,Y 392.3,Z 425.761,A -85,B 0,C 180,E1 -11595.075,E2 -11595.075} C_VEL
LIN {X 0,Y 391.483,Z 436.698,A -85,B 0,C 180,E1 -11596.288,E2 -11596.288} C_VEL
LIN {X 0,Y 390.754,Z 445.761,A -85,B 0,C 180,E1 -11597.534,E2 -11597.534} C_VEL
LIN {X 0,Y 389.951,Z 454.875,A -85,B 0,C 180,E1 -11599.09,E2 -11599.09} C_VEL
LIN {X 0,Y 389.436,Z 462.216,A -85,B 0,C 180,E1 -11600.651,E2 -11600.651} C_VEL
LIN {X 0,Y 389.049,Z 468.088,A -85,B 0,C 180,E1 -11602.212,E2 -11602.212} C_VEL
LIN {X 0,Y 388.787,Z 472.903,A -85,B 0,C 180,E1 -11603.853,E2 -11603.853} C_VEL
LIN {X 0,Y 388.757,Z 475.129,A -85,B 0,C 180,E1 -11604.812,E2 -11604.812} C_VEL
LIN {X 0,Y 388.698,Z 477.114,A -85,B 0,C 180,E1 -11605.851,E2 -11605.851} C_VEL
LIN {X 0,Y 388.606,Z 478.681,A -85,B 0,C 180,E1 -11606.888,E2 -11606.888} C_VEL
LIN {X 0,Y 388.622,Z 479.816,A -85,B 0,C 180,E1 -11607.926,E2 -11607.926} C_VEL
LIN {X 0,Y 388.66,Z 480.524,A -85,B 0,C 180,E1 -11608.962,E2 -11608.962} C_VEL
LIN {X 0,Y 388.677,Z 480.845,A -85,B 0,C 180,E1 -11609.998,E2 -11609.998} C_VEL
LIN {X 0,Y 388.66,Z 480.78,A -85,B 0,C 180,E1 -11611.034,E2 -11611.034} C_VEL
LIN {X 0,Y 388.62,Z 480.309,A -85,B 0,C 180,E1 -11612.071,E2 -11612.071} C_VEL
LIN {X 0,Y 388.703,Z 478.125,A -85,B 0,C 180,E1 -11614.146,E2 -11614.146} C_VEL
LIN {X 0,Y 388.8,Z 475.12,A -85,B 0,C 180,E1 -11615.841,E2 -11615.841} C_VEL
LIN {X 0,Y 389.111,Z 470.2,A -85,B 0,C 180,E1 -11617.784,E2 -11617.784} C_VEL
LIN {X 0,Y 389.641,Z 463.944,A -85,B 0,C 180,E1 -11619.603,E2 -11619.603} C_VEL
LIN {X 0,Y 390.27,Z 457.145,A -85,B 0,C 180,E1 -11621.16,E2 -11621.16} C_VEL
LIN {X 0,Y 391.213,Z 448.689,A -85,B 0,C 180,E1 -11622.711,E2 -11622.711} C_VEL
LIN {X 0,Y 392.093,Z 440.004,A -85,B 0,C 180,E1 -11624.002,E2 -11624.002} C_VEL
LIN {X 0,Y 393.06,Z 429.133,A -85,B 0,C 180,E1 -11625.313,E2 -11625.313} C_VEL
LIN {X 0,Y 394.031,Z 418.727,A -85,B 0,C 180,E1 -11626.313,E2 -11626.313} C_VEL
LIN {X 0,Y 395.022,Z 406.875,A -85,B 0,C 180,E1 -11627.203,E2 -11627.203} C_VEL
LIN {X 0,Y 395.818,Z 394.62,A -85,B 0,C 180,E1 -11627.9,E2 -11627.9} C_VEL
LIN {X 0,Y 396.488,Z 382.078,A -85,B 0,C 180,E1 -11628.403,E2 -11628.403} C_VEL
LIN {X 0,Y 396.895,Z 368.678,A -85,B 0,C 180,E1 -11628.728,E2 -11628.728} C_VEL
LIN {X 0,Y 397.937,Z 296.657,A -85,B 0,C 180,E1 -11630.076,E2 -11630.076} C_VEL
LIN {X 0,Y 394.424,Z 276.983,A -85,B 0,C 180,E1 -11630.684,E2 -11630.684} C_VEL
LIN {X 0,Y 392.748,Z 268.709,A -85,B 0,C 180,E1 -11630.993,E2 -11630.993} C_VEL
LIN {X 0,Y 393.673,Z 256.58,A -85,B 0,C 180,E1 -11633.681,E2 -11633.681} C_VEL
LIN {X 0,Y 392.514,Z 249.444,A -85,B 0,C 180,E1 -11635.448,E2 -11635.448} C_VEL
LIN {X 0,Y 390.159,Z 238.67,A -85,B 0,C 180,E1 -11638.268,E2 -11638.268} C_VEL
LIN {X 0,Y 390.097,Z 238.393,A -85,B 0,C 180,E1 -11638.515,E2 -11638.515} C_VEL
LIN {X 0,Y 390.035,Z 238.398,A -85,B 0,C 180,E1 -11642.121,E2 -11642.121} C_VEL
LIN {X 0,Y 390.088,Z 238.387,A -85,B 0,C 180,E1 -11645.204,E2 -11645.204} C_VEL
LIN {X 0,Y 390.067,Z 238.392,A -85,B 0,C 180,E1 -11649.093,E2 -11649.093} C_VEL
LIN {X 0,Y 390.039,Z 238.391,A -85,B 0,C 180,E1 -11652.37,E2 -11652.37} C_VEL
LIN {X 0,Y 390.044,Z 238.395,A -85,B 0,C 180,E1 -11655.351,E2 -11655.351} C_VEL
LIN {X 0,Y 390.02,Z 238.396,A -85,B 0,C 180,E1 -11658.182,E2 -11658.182} C_VEL
LIN {X 0,Y 390.057,Z 238.395,A -85,B 0,C 180,E1 -11660.9,E2 -11660.9} C_VEL
LIN {X 0,Y 390.083,Z 238.396,A -85,B 0,C 180,E1 -11664.79,E2 -11664.79} C_VEL
LIN {X 0,Y 390.021,Z 238.402,A -85,B 0,C 180,E1 -11668.492,E2 -11668.492} C_VEL
LIN {X 0,Y 390.028,Z 238.398,A -85,B 0,C 180,E1 -11672.06,E2 -11672.06} C_VEL
LIN {X 0,Y 390.038,Z 238.397,A -85,B 0,C 180,E1 -11675.513,E2 -11675.513} C_VEL
LIN {X 0,Y 390.049,Z 238.393,A -85,B 0,C 180,E1 -11678.874,E2 -11678.874} C_VEL
LIN {X 0,Y 390.104,Z 238.387,A -85,B 0,C 180,E1 -11682.162,E2 -11682.162} C_VEL
LIN {X 0,Y 390.134,Z 238.389,A -85,B 0,C 180,E1 -11685.389,E2 -11685.389} C_VEL
LIN {X 0,Y 390.133,Z 238.38,A -85,B 0,C 180,E1 -11688.567,E2 -11688.567} C_VEL
LIN {X 0,Y 390.255,Z 238.362,A -85,B 0,C 180,E1 -11692.072,E2 -11692.072} C_VEL
LIN {X 0,Y 390.195,Z 238.379,A -85,B 0,C 180,E1 -11694.829,E2 -11694.829} C_VEL
LIN {X 0,Y 390.388,Z 238.355,A -85,B 0,C 180,E1 -11697.933,E2 -11697.933} C_VEL
LIN {X 0,Y 390.392,Z 238.354,A -85,B 0,C 180,E1 -11702.059,E2 -11702.059} C_VEL
LIN {X 0,Y 390.237,Z 238.372,A -85,B 0,C 180,E1 -11706.46,E2 -11706.46} C_VEL
LIN {X 0,Y 390.174,Z 238.379,A -85,B 0,C 180,E1 -11709.325,E2 -11709.325} C_VEL
LIN {X 0,Y 390.15,Z 238.381,A -85,B 0,C 180,E1 -11712.479,E2 -11712.479} C_VEL
LIN {X 0,Y 390.116,Z 238.392,A -85,B 0,C 180,E1 -11715.673,E2 -11715.673} C_VEL
LIN {X 0,Y 390.078,Z 238.392,A -85,B 0,C 180,E1 -11718.918,E2 -11718.918} C_VEL
LIN {X 0,Y 390.011,Z 238.402,A -85,B 0,C 180,E1 -11722.231,E2 -11722.231} C_VEL
LIN {X 0,Y 390.091,Z 238.39,A -85,B 0,C 180,E1 -11725.739,E2 -11725.739} C_VEL
LIN {X 0,Y 390.029,Z 238.392,A -85,B 0,C 180,E1 -11729.106,E2 -11729.106} C_VEL
LIN {X 0,Y 390.012,Z 238.396,A -85,B 0,C 180,E1 -11732.718,E2 -11732.718} C_VEL
LIN {X 0,Y 390.025,Z 238.395,A -85,B 0,C 180,E1 -11735.822,E2 -11735.822} C_VEL
LIN {X 0,Y 390.041,Z 238.402,A -85,B 0,C 180,E1 -11739.216,E2 -11739.216} C_VEL
LIN {X 0,Y 390.114,Z 238.552,A -85,B 0,C 180,E1 -11742.968,E2 -11742.968} C_VEL
LIN {X 0,Y 392.351,Z 249.126,A -85,B 0,C 180,E1 -11745.758,E2 -11745.758} C_VEL
LIN {X 0,Y 393.168,Z 254.603,A -85,B 0,C 180,E1 -11747.121,E2 -11747.121} C_VEL
LIN {X 0,Y 392.923,Z 259.005,A -85,B 0,C 180,E1 -11748.071,E2 -11748.071} C_VEL
LIN {X 0,Y 397.094,Z 278.03,A -85,B 0,C 180,E1 -11748.743,E2 -11748.743} C_VEL
LIN {X 0,Y 398.192,Z 285.045,A -85,B 0,C 180,E1 -11748.949,E2 -11748.949} C_VEL
LIN {X 0,Y 396.777,Z 367.048,A -85,B 0,C 180,E1 -11750.503,E2 -11750.503} C_VEL
LIN {X 0,Y 396.152,Z 380.766,A -85,B 0,C 180,E1 -11750.98,E2 -11750.98} C_VEL
LIN {X 0,Y 395.454,Z 393.092,A -85,B 0,C 180,E1 -11751.62,E2 -11751.62} C_VEL
LIN {X 0,Y 394.636,Z 404.452,A -85,B 0,C 180,E1 -11752.416,E2 -11752.416} C_VEL
LIN {X 0,Y 393.64,Z 415.941,A -85,B 0,C 180,E1 -11753.449,E2 -11753.449} C_VEL
LIN {X 0,Y 392.636,Z 426.088,A -85,B 0,C 180,E1 -11754.587,E2 -11754.587} C_VEL
LIN {X 0,Y 391.638,Z 436.03,A -85,B 0,C 180,E1 -11755.984,E2 -11755.984} C_VEL
LIN {X 0,Y 390.844,Z 443.946,A -85,B 0,C 180,E1 -11757.356,E2 -11757.356} C_VEL
LIN {X 0,Y 390.024,Z 452.054,A -85,B 0,C 180,E1 -11759.101,E2 -11759.101} C_VEL
LIN {X 0,Y 389.475,Z 458.305,A -85,B 0,C 180,E1 -11760.845,E2 -11760.845} C_VEL
LIN {X 0,Y 389.043,Z 463.341,A -85,B 0,C 180,E1 -11762.693,E2 -11762.693} C_VEL
LIN {X 0,Y 388.737,Z 466.502,A -85,B 0,C 180,E1 -11764.287,E2 -11764.287} C_VEL
LIN {X 0,Y 388.582,Z 468.152,A -85,B 0,C 180,E1 -11765.421,E2 -11765.421} C_VEL
LIN {X 0,Y 388.44,Z 469.761,A -85,B 0,C 180,E1 -11767.314,E2 -11767.314} C_VEL
LIN {X 0,Y 388.381,Z 470.131,A -85,B 0,C 180,E1 -11768.784,E2 -11768.784} C_VEL
LIN {X 0,Y 388.454,Z 469.718,A -85,B 0,C 180,E1 -11770.167,E2 -11770.167} C_VEL
LIN {X 0,Y 388.503,Z 467.996,A -85,B 0,C 180,E1 -11772.091,E2 -11772.091} C_VEL
LIN {X 0,Y 388.677,Z 466.013,A -85,B 0,C 180,E1 -11773.381,E2 -11773.381} C_VEL
LIN {X 0,Y 388.951,Z 461.72,A -85,B 0,C 180,E1 -11775.349,E2 -11775.349} C_VEL
LIN {X 0,Y 389.257,Z 456.304,A -85,B 0,C 180,E1 -11777.124,E2 -11777.124} C_VEL
LIN {X 0,Y 389.781,Z 449.592,A -85,B 0,C 180,E1 -11778.825,E2 -11778.825} C_VEL
LIN {X 0,Y 390.344,Z 441.658,A -85,B 0,C 180,E1 -11780.415,E2 -11780.415} C_VEL
LIN {X 0,Y 391.081,Z 433.486,A -85,B 0,C 180,E1 -11781.736,E2 -11781.736} C_VEL
LIN {X 0,Y 391.839,Z 423.548,A -85,B 0,C 180,E1 -11783.048,E2 -11783.048} C_VEL
LIN {X 0,Y 392.677,Z 413.731,A -85,B 0,C 180,E1 -11784.095,E2 -11784.095} C_VEL
LIN {X 0,Y 393.393,Z 403.192,A -85,B 0,C 180,E1 -11785.005,E2 -11785.005} C_VEL
LIN {X 0,Y 394.049,Z 390.556,A -85,B 0,C 180,E1 -11785.847,E2 -11785.847} C_VEL
LIN {X 0,Y 394.694,Z 377.676,A -85,B 0,C 180,E1 -11786.467,E2 -11786.467} C_VEL
LIN {X 0,Y 395.06,Z 364.627,A -85,B 0,C 180,E1 -11786.879,E2 -11786.879} C_VEL
LIN {X 0,Y 395.855,Z 307.008,A -85,B 0,C 180,E1 -11787.952,E2 -11787.952} C_VEL
LIN {X 0,Y 395.337,Z 301.178,A -85,B 0,C 180,E1 -11788.085,E2 -11788.085} C_VEL
LIN {X 0,Y 392.898,Z 291.774,A -85,B 0,C 180,E1 -11788.371,E2 -11788.371} C_VEL
LIN {X 0,Y 388.133,Z 276.834,A -85,B 0,C 180,E1 -11788.867,E2 -11788.867} C_VEL
LIN {X 0,Y 385.147,Z 259.526,A -85,B 0,C 180,E1 -11789.359,E2 -11789.359} C_VEL
LIN {X 0,Y 385.126,Z 258.618,A -85,B 0,C 180,E1 -11789.479,E2 -11789.479} C_VEL
LIN {X 0,Y 385.531,Z 252.012,A -85,B 0,C 180,E1 -11791.046,E2 -11791.046} C_VEL
LIN {X 0,Y 383.801,Z 242.859,A -85,B 0,C 180,E1 -11793.413,E2 -11793.413} C_VEL
LIN {X 0,Y 383.079,Z 239.343,A -85,B 0,C 180,E1 -11794.408,E2 -11794.408} C_VEL
LIN {X 0,Y 383.214,Z 239.253,A -85,B 0,C 180,E1 -11797.377,E2 -11797.377} C_VEL
LIN {X 0,Y 383.097,Z 239.26,A -85,B 0,C 180,E1 -11800.572,E2 -11800.572} C_VEL
LIN {X 0,Y 383.089,Z 239.267,A -85,B 0,C 180,E1 -11803.799,E2 -11803.799} C_VEL
LIN {X 0,Y 383.058,Z 239.269,A -85,B 0,C 180,E1 -11807.457,E2 -11807.457} C_VEL
LIN {X 0,Y 382.993,Z 239.274,A -85,B 0,C 180,E1 -11810.65,E2 -11810.65} C_VEL
LIN {X 0,Y 382.979,Z 239.28,A -85,B 0,C 180,E1 -11813.812,E2 -11813.812} C_VEL
LIN {X 0,Y 382.959,Z 239.278,A -85,B 0,C 180,E1 -11817.311,E2 -11817.311} C_VEL
LIN {X 0,Y 382.95,Z 239.279,A -85,B 0,C 180,E1 -11820.923,E2 -11820.923} C_VEL
LIN {X 0,Y 382.982,Z 239.278,A -85,B 0,C 180,E1 -11824.673,E2 -11824.673} C_VEL
LIN {X 0,Y 382.965,Z 239.278,A -85,B 0,C 180,E1 -11827.907,E2 -11827.907} C_VEL
LIN {X 0,Y 382.936,Z 239.281,A -85,B 0,C 180,E1 -11831.355,E2 -11831.355} C_VEL
LIN {X 0,Y 382.966,Z 239.28,A -85,B 0,C 180,E1 -11834.307,E2 -11834.307} C_VEL
LIN {X 0,Y 382.991,Z 239.276,A -85,B 0,C 180,E1 -11837.245,E2 -11837.245} C_VEL
LIN {X 0,Y 382.968,Z 239.279,A -85,B 0,C 180,E1 -11840.424,E2 -11840.424} C_VEL
LIN {X 0,Y 382.999,Z 239.272,A -85,B 0,C 180,E1 -11844.048,E2 -11844.048} C_VEL
LIN {X 0,Y 382.971,Z 239.278,A -85,B 0,C 180,E1 -11847.584,E2 -11847.584} C_VEL
LIN {X 0,Y 382.964,Z 239.277,A -85,B 0,C 180,E1 -11850.304,E2 -11850.304} C_VEL
LIN {X 0,Y 382.994,Z 239.274,A -85,B 0,C 180,E1 -11854.05,E2 -11854.05} C_VEL
LIN {X 0,Y 382.981,Z 239.281,A -85,B 0,C 180,E1 -11857.339,E2 -11857.339} C_VEL
LIN {X 0,Y 383.054,Z 239.266,A -85,B 0,C 180,E1 -11860.721,E2 -11860.721} C_VEL
LIN {X 0,Y 383.077,Z 239.266,A -85,B 0,C 180,E1 -11864.031,E2 -11864.031} C_VEL
LIN {X 0,Y 383.134,Z 239.258,A -85,B 0,C 180,E1 -11867.289,E2 -11867.289} C_VEL
LIN {X 0,Y 383.139,Z 239.256,A -85,B 0,C 180,E1 -11870.502,E2 -11870.502} C_VEL
LIN {X 0,Y 383.237,Z 239.247,A -85,B 0,C 180,E1 -11873.687,E2 -11873.687} C_VEL
LIN {X 0,Y 383.379,Z 239.23,A -85,B 0,C 180,E1 -11877.903,E2 -11877.903} C_VEL
LIN {X 0,Y 383.375,Z 239.232,A -85,B 0,C 180,E1 -11882.105,E2 -11882.105} C_VEL
LIN {X 0,Y 383.243,Z 239.249,A -85,B 0,C 180,E1 -11886.321,E2 -11886.321} C_VEL
LIN {X 0,Y 383.149,Z 239.254,A -85,B 0,C 180,E1 -11889.506,E2 -11889.506} C_VEL
LIN {X 0,Y 383.139,Z 239.255,A -85,B 0,C 180,E1 -11893.539,E2 -11893.539} C_VEL
LIN {X 0,Y 383.108,Z 239.262,A -85,B 0,C 180,E1 -11897.072,E2 -11897.072} C_VEL
LIN {X 0,Y 383.044,Z 239.272,A -85,B 0,C 180,E1 -11900.649,E2 -11900.649} C_VEL
LIN {X 0,Y 383.025,Z 239.269,A -85,B 0,C 180,E1 -11903.811,E2 -11903.811} C_VEL
LIN {X 0,Y 382.985,Z 239.278,A -85,B 0,C 180,E1 -11907.311,E2 -11907.311} C_VEL
LIN {X 0,Y 382.997,Z 239.277,A -85,B 0,C 180,E1 -11910.921,E2 -11910.921} C_VEL
LIN {X 0,Y 383.033,Z 239.269,A -85,B 0,C 180,E1 -11914.67,E2 -11914.67} C_VEL
LIN {X 0,Y 383.01,Z 239.273,A -85,B 0,C 180,E1 -11917.904,E2 -11917.904} C_VEL
LIN {X 0,Y 382.977,Z 239.281,A -85,B 0,C 180,E1 -11921.352,E2 -11921.352} C_VEL
LIN {X 0,Y 383.004,Z 239.272,A -85,B 0,C 180,E1 -11924.303,E2 -11924.303} C_VEL
LIN {X 0,Y 382.998,Z 239.275,A -85,B 0,C 180,E1 -11927.237,E2 -11927.237} C_VEL
LIN {X 0,Y 383.002,Z 239.273,A -85,B 0,C 180,E1 -11930.42,E2 -11930.42} C_VEL
LIN {X 0,Y 383.04,Z 239.273,A -85,B 0,C 180,E1 -11934.044,E2 -11934.044} C_VEL
LIN {X 0,Y 383.003,Z 239.274,A -85,B 0,C 180,E1 -11937.578,E2 -11937.578} C_VEL
LIN {X 0,Y 382.996,Z 239.279,A -85,B 0,C 180,E1 -11940.299,E2 -11940.299} C_VEL
LIN {X 0,Y 383.081,Z 239.388,A -85,B 0,C 180,E1 -11942.627,E2 -11942.627} C_VEL
LIN {X 0,Y 384.787,Z 248.197,A -85,B 0,C 180,E1 -11944.87,E2 -11944.87} C_VEL
LIN {X 0,Y 385.888,Z 254.425,A -85,B 0,C 180,E1 -11946.378,E2 -11946.378} C_VEL
LIN {X 0,Y 385.068,Z 266.623,A -85,B 0,C 180,E1 -11949.15,E2 -11949.15} C_VEL
LIN {X 0,Y 384.939,Z 269.249,A -85,B 0,C 180,E1 -11949.649,E2 -11949.649} C_VEL
LIN {X 0,Y 389.336,Z 297.682,A -85,B 0,C 180,E1 -11950.433,E2 -11950.433} C_VEL
LIN {X 0,Y 388.164,Z 377.138,A -85,B 0,C 180,E1 -11951.936,E2 -11951.936} C_VEL
LIN {X 0,Y 387.593,Z 391,A -85,B 0,C 180,E1 -11952.42,E2 -11952.42} C_VEL
LIN {X 0,Y 386.886,Z 403.963,A -85,B 0,C 180,E1 -11953.102,E2 -11953.102} C_VEL
LIN {X 0,Y 385.999,Z 416.558,A -85,B 0,C 180,E1 -11954.013,E2 -11954.013} C_VEL
LIN {X 0,Y 385.168,Z 427.795,A -85,B 0,C 180,E1 -11955.063,E2 -11955.063} C_VEL
LIN {X 0,Y 384.398,Z 437.888,A -85,B 0,C 180,E1 -11956.249,E2 -11956.249} C_VEL
LIN {X 0,Y 383.617,Z 447.01,A -85,B 0,C 180,E1 -11957.567,E2 -11957.567} C_VEL
LIN {X 0,Y 382.855,Z 455.901,A -85,B 0,C 180,E1 -11959.153,E2 -11959.153} C_VEL
LIN {X 0,Y 382.323,Z 463.011,A -85,B 0,C 180,E1 -11960.742,E2 -11960.742} C_VEL
LIN {X 0,Y 381.88,Z 469.489,A -85,B 0,C 180,E1 -11962.597,E2 -11962.597} C_VEL
LIN {X 0,Y 381.701,Z 473.024,A -85,B 0,C 180,E1 -11963.878,E2 -11963.878} C_VEL
LIN {X 0,Y 381.625,Z 476.938,A -85,B 0,C 180,E1 -11965.774,E2 -11965.774} C_VEL
LIN {X 0,Y 381.52,Z 478.519,A -85,B 0,C 180,E1 -11966.83,E2 -11966.83} C_VEL
LIN {X 0,Y 381.52,Z 479.682,A -85,B 0,C 180,E1 -11967.887,E2 -11967.887} C_VEL
LIN {X 0,Y 381.559,Z 480.405,A -85,B 0,C 180,E1 -11968.943,E2 -11968.943} C_VEL
LIN {X 0,Y 381.578,Z 480.74,A -85,B 0,C 180,E1 -11969.998,E2 -11969.998} C_VEL
LIN {X 0,Y 381.558,Z 480.688,A -85,B 0,C 180,E1 -11971.054,E2 -11971.054} C_VEL
LIN {X 0,Y 381.518,Z 480.242,A -85,B 0,C 180,E1 -11972.11,E2 -11972.11} C_VEL
LIN {X 0,Y 381.633,Z 478.088,A -85,B 0,C 180,E1 -11974.223,E2 -11974.223} C_VEL
LIN {X 0,Y 381.749,Z 474.626,A -85,B 0,C 180,E1 -11976.189,E2 -11976.189} C_VEL
LIN {X 0,Y 382.07,Z 470.235,A -85,B 0,C 180,E1 -11977.928,E2 -11977.928} C_VEL
LIN {X 0,Y 382.612,Z 464.012,A -85,B 0,C 180,E1 -11979.781,E2 -11979.781} C_VEL
LIN {X 0,Y 383.29,Z 457.25,A -85,B 0,C 180,E1 -11981.366,E2 -11981.366} C_VEL
LIN {X 0,Y 384.3,Z 448.87,A -85,B 0,C 180,E1 -11982.944,E2 -11982.944} C_VEL
LIN {X 0,Y 385.212,Z 440.264,A -85,B 0,C 180,E1 -11984.257,E2 -11984.257} C_VEL
LIN {X 0,Y 386.225,Z 429.652,A -85,B 0,C 180,E1 -11985.572,E2 -11985.572} C_VEL
LIN {X 0,Y 387.246,Z 419.216,A -85,B 0,C 180,E1 -11986.607,E2 -11986.607} C_VEL
LIN {X 0,Y 388.287,Z 407.614,A -85,B 0,C 180,E1 -11987.511,E2 -11987.511} C_VEL
LIN {X 0,Y 389.205,Z 394.328,A -85,B 0,C 180,E1 -11988.283,E2 -11988.283} C_VEL
LIN {X 0,Y 389.891,Z 381.701,A -85,B 0,C 180,E1 -11988.795,E2 -11988.795} C_VEL
LIN {X 0,Y 390.326,Z 368.298,A -85,B 0,C 180,E1 -11989.119,E2 -11989.119} C_VEL
LIN {X 0,Y 391.415,Z 297.533,A -85,B 0,C 180,E1 -11990.466,E2 -11990.466} C_VEL
LIN {X 0,Y 387.889,Z 277.915,A -85,B 0,C 180,E1 -11991.09,E2 -11991.09} C_VEL
LIN {X 0,Y 385.925,Z 268.63,A -85,B 0,C 180,E1 -11991.448,E2 -11991.448} C_VEL
LIN {X 0,Y 386.796,Z 258.099,A -85,B 0,C 180,E1 -11993.814,E2 -11993.814} C_VEL
LIN {X 0,Y 385.583,Z 250.84,A -85,B 0,C 180,E1 -11995.649,E2 -11995.649} C_VEL
LIN {X 0,Y 383.126,Z 239.652,A -85,B 0,C 180,E1 -11998.633,E2 -11998.633} C_VEL
LIN {X 0,Y 383.045,Z 239.271,A -85,B 0,C 180,E1 -11998.94,E2 -11998.94} C_VEL
LIN {X 0,Y 382.991,Z 239.274,A -85,B 0,C 180,E1 -12002.419,E2 -12002.419} C_VEL
LIN {X 0,Y 383.027,Z 239.27,A -85,B 0,C 180,E1 -12005.953,E2 -12005.953} C_VEL
LIN {X 0,Y 382.997,Z 239.275,A -85,B 0,C 180,E1 -12009.58,E2 -12009.58} C_VEL
LIN {X 0,Y 383.008,Z 239.269,A -85,B 0,C 180,E1 -12012.775,E2 -12012.775} C_VEL
LIN {X 0,Y 382.997,Z 239.269,A -85,B 0,C 180,E1 -12015.786,E2 -12015.786} C_VEL
LIN {X 0,Y 382.964,Z 239.282,A -85,B 0,C 180,E1 -12018.797,E2 -12018.797} C_VEL
LIN {X 0,Y 382.993,Z 239.277,A -85,B 0,C 180,E1 -12022.094,E2 -12022.094} C_VEL
LIN {X 0,Y 383.017,Z 239.273,A -85,B 0,C 180,E1 -12025.329,E2 -12025.329} C_VEL
LIN {X 0,Y 382.98,Z 239.279,A -85,B 0,C 180,E1 -12029.078,E2 -12029.078} C_VEL
LIN {X 0,Y 382.983,Z 239.281,A -85,B 0,C 180,E1 -12032.689,E2 -12032.689} C_VEL
LIN {X 0,Y 383.006,Z 239.273,A -85,B 0,C 180,E1 -12036.187,E2 -12036.187} C_VEL
LIN {X 0,Y 383.05,Z 239.266,A -85,B 0,C 180,E1 -12039.595,E2 -12039.595} C_VEL
LIN {X 0,Y 383.087,Z 239.26,A -85,B 0,C 180,E1 -12042.927,E2 -12042.927} C_VEL
LIN {X 0,Y 383.117,Z 239.26,A -85,B 0,C 180,E1 -12046.46,E2 -12046.46} C_VEL
LIN {X 0,Y 383.129,Z 239.259,A -85,B 0,C 180,E1 -12050.494,E2 -12050.494} C_VEL
LIN {X 0,Y 383.247,Z 239.246,A -85,B 0,C 180,E1 -12053.679,E2 -12053.679} C_VEL
LIN {X 0,Y 383.354,Z 239.232,A -85,B 0,C 180,E1 -12057.895,E2 -12057.895} C_VEL
LIN {X 0,Y 383.358,Z 239.23,A -85,B 0,C 180,E1 -12062.097,E2 -12062.097} C_VEL
LIN {X 0,Y 383.203,Z 239.248,A -85,B 0,C 180,E1 -12066.448,E2 -12066.448} C_VEL
LIN {X 0,Y 383.124,Z 239.257,A -85,B 0,C 180,E1 -12069.498,E2 -12069.498} C_VEL
LIN {X 0,Y 383.105,Z 239.258,A -85,B 0,C 180,E1 -12073.532,E2 -12073.532} C_VEL
LIN {X 0,Y 383.071,Z 239.262,A -85,B 0,C 180,E1 -12077.065,E2 -12077.065} C_VEL
LIN {X 0,Y 383.004,Z 239.276,A -85,B 0,C 180,E1 -12080.643,E2 -12080.643} C_VEL
LIN {X 0,Y 382.996,Z 239.277,A -85,B 0,C 180,E1 -12083.804,E2 -12083.804} C_VEL
LIN {X 0,Y 383.052,Z 239.27,A -85,B 0,C 180,E1 -12086.12,E2 -12086.12} C_VEL
LIN {X 0,Y 382.962,Z 239.275,A -85,B 0,C 180,E1 -12089.696,E2 -12089.696} C_VEL
LIN {X 0,Y 382.972,Z 239.278,A -85,B 0,C 180,E1 -12093.397,E2 -12093.397} C_VEL
LIN {X 0,Y 383.002,Z 239.271,A -85,B 0,C 180,E1 -12096.162,E2 -12096.162} C_VEL
LIN {X 0,Y 382.987,Z 239.279,A -85,B 0,C 180,E1 -12099.954,E2 -12099.954} C_VEL
LIN {X 0,Y 383.085,Z 239.415,A -85,B 0,C 180,E1 -12102.563,E2 -12102.563} C_VEL
LIN {X 0,Y 385.257,Z 249.702,A -85,B 0,C 180,E1 -12105.345,E2 -12105.345} C_VEL
LIN {X 0,Y 386.306,Z 256.126,A -85,B 0,C 180,E1 -12106.985,E2 -12106.985} C_VEL
LIN {X 0,Y 386.171,Z 259.178,A -85,B 0,C 180,E1 -12107.626,E2 -12107.626} C_VEL
LIN {X 0,Y 390.616,Z 279.189,A -85,B 0,C 180,E1 -12108.353,E2 -12108.353} C_VEL
LIN {X 0,Y 391.67,Z 284.946,A -85,B 0,C 180,E1 -12108.536,E2 -12108.536} C_VEL
LIN {X 0,Y 390.191,Z 366.714,A -85,B 0,C 180,E1 -12110.107,E2 -12110.107} C_VEL
LIN {X 0,Y 389.629,Z 379.851,A -85,B 0,C 180,E1 -12110.563,E2 -12110.563} C_VEL
LIN {X 0,Y 388.9,Z 391.984,A -85,B 0,C 180,E1 -12111.184,E2 -12111.184} C_VEL
LIN {X 0,Y 388.037,Z 403.685,A -85,B 0,C 180,E1 -12111.993,E2 -12111.993} C_VEL
LIN {X 0,Y 386.984,Z 415.243,A -85,B 0,C 180,E1 -12113.033,E2 -12113.033} C_VEL
LIN {X 0,Y 385.888,Z 425.551,A -85,B 0,C 180,E1 -12114.194,E2 -12114.194} C_VEL
LIN {X 0,Y 384.91,Z 435.093,A -85,B 0,C 180,E1 -12115.529,E2 -12115.529} C_VEL
LIN {X 0,Y 383.937,Z 444.077,A -85,B 0,C 180,E1 -12117.102,E2 -12117.102} C_VEL
LIN {X 0,Y 383.083,Z 451.789,A -85,B 0,C 180,E1 -12118.786,E2 -12118.786} C_VEL
LIN {X 0,Y 382.571,Z 457.197,A -85,B 0,C 180,E1 -12120.266,E2 -12120.266} C_VEL
LIN {X 0,Y 382.142,Z 462.113,A -85,B 0,C 180,E1 -12121.966,E2 -12121.966} C_VEL
LIN {X 0,Y 381.742,Z 465.974,A -85,B 0,C 180,E1 -12123.78,E2 -12123.78} C_VEL
LIN {X 0,Y 381.56,Z 467.759,A -85,B 0,C 180,E1 -12124.937,E2 -12124.937} C_VEL
LIN {X 0,Y 381.41,Z 469.072,A -85,B 0,C 180,E1 -12126.087,E2 -12126.087} C_VEL
LIN {X 0,Y 381.354,Z 469.859,A -85,B 0,C 180,E1 -12127.233,E2 -12127.233} C_VEL
LIN {X 0,Y 381.285,Z 470.199,A -85,B 0,C 180,E1 -12128.37,E2 -12128.37} C_VEL
LIN {X 0,Y 381.343,Z 469.874,A -85,B 0,C 180,E1 -12130.018,E2 -12130.018} C_VEL
LIN {X 0,Y 381.402,Z 468.493,A -85,B 0,C 180,E1 -12131.746,E2 -12131.746} C_VEL
LIN {X 0,Y 381.564,Z 466.358,A -85,B 0,C 180,E1 -12133.27,E2 -12133.27} C_VEL
LIN {X 0,Y 381.8,Z 462.681,A -85,B 0,C 180,E1 -12135.068,E2 -12135.068} C_VEL
LIN {X 0,Y 382.128,Z 458.187,A -85,B 0,C 180,E1 -12136.685,E2 -12136.685} C_VEL
LIN {X 0,Y 382.522,Z 452.295,A -85,B 0,C 180,E1 -12138.342,E2 -12138.342} C_VEL
LIN {X 0,Y 383.078,Z 444.971,A -85,B 0,C 180,E1 -12139.965,E2 -12139.965} C_VEL
LIN {X 0,Y 383.887,Z 435.825,A -85,B 0,C 180,E1 -12141.58,E2 -12141.58} C_VEL
LIN {X 0,Y 384.638,Z 426.433,A -85,B 0,C 180,E1 -12142.917,E2 -12142.917} C_VEL
LIN {X 0,Y 385.557,Z 415.885,A -85,B 0,C 180,E1 -12144.117,E2 -12144.117} C_VEL
LIN {X 0,Y 386.419,Z 404.193,A -85,B 0,C 180,E1 -12145.176,E2 -12145.176} C_VEL
LIN {X 0,Y 387.115,Z 392.643,A -85,B 0,C 180,E1 -12145.989,E2 -12145.989} C_VEL
LIN {X 0,Y 387.764,Z 379.242,A -85,B 0,C 180,E1 -12146.674,E2 -12146.674} C_VEL
LIN {X 0,Y 388.218,Z 366.303,A -85,B 0,C 180,E1 -12147.116,E2 -12147.116} C_VEL
LIN {X 0,Y 389.353,Z 283.481,A -85,B 0,C 180,E1 -12148.685,E2 -12148.685} C_VEL
LIN {X 0,Y 388.133,Z 276.834,A -85,B 0,C 180,E1 -12148.867,E2 -12148.867} C_VEL
LIN {X 0,Y 386.231,Z 271.739,A -85,B 0,C 180,E1 -12149.077,E2 -12149.077} C_VEL
LIN {X 0,Y 378.398,Z 259.61,A -85,B 0,C 180,E1 -12149.681,E2 -12149.681} C_VEL
LIN {X 0,Y 378.214,Z 258.952,A -85,B 0,C 180,E1 -12149.759,E2 -12149.759} C_VEL
LIN {X 0,Y 378.551,Z 253.48,A -85,B 0,C 180,E1 -12151.065,E2 -12151.065} C_VEL
LIN {X 0,Y 377.07,Z 245.309,A -85,B 0,C 180,E1 -12153.207,E2 -12153.207} C_VEL
LIN {X 0,Y 376.078,Z 240.183,A -85,B 0,C 180,E1 -12154.658,E2 -12154.658} C_VEL
LIN {X 0,Y 376.168,Z 240.13,A -85,B 0,C 180,E1 -12157.516,E2 -12157.516} C_VEL
LIN {X 0,Y 376.049,Z 240.139,A -85,B 0,C 180,E1 -12160.773,E2 -12160.773} C_VEL
LIN {X 0,Y 376.028,Z 240.144,A -85,B 0,C 180,E1 -12164.064,E2 -12164.064} C_VEL
LIN {X 0,Y 376.006,Z 240.149,A -85,B 0,C 180,E1 -12167.61,E2 -12167.61} C_VEL
LIN {X 0,Y 375.944,Z 240.151,A -85,B 0,C 180,E1 -12170.836,E2 -12170.836} C_VEL
LIN {X 0,Y 375.928,Z 240.157,A -85,B 0,C 180,E1 -12174.288,E2 -12174.288} C_VEL
LIN {X 0,Y 375.901,Z 240.161,A -85,B 0,C 180,E1 -12177.868,E2 -12177.868} C_VEL
LIN {X 0,Y 375.923,Z 240.156,A -85,B 0,C 180,E1 -12180.697,E2 -12180.697} C_VEL
LIN {X 0,Y 375.928,Z 240.158,A -85,B 0,C 180,E1 -12184.116,E2 -12184.116} C_VEL
LIN {X 0,Y 375.92,Z 240.158,A -85,B 0,C 180,E1 -12186.747,E2 -12186.747} C_VEL
LIN {X 0,Y 375.912,Z 240.157,A -85,B 0,C 180,E1 -12189.966,E2 -12189.966} C_VEL
LIN {X 0,Y 375.902,Z 240.157,A -85,B 0,C 180,E1 -12193.772,E2 -12193.772} C_VEL
LIN {X 0,Y 375.914,Z 240.162,A -85,B 0,C 180,E1 -12196.816,E2 -12196.816} C_VEL
LIN {X 0,Y 375.917,Z 240.158,A -85,B 0,C 180,E1 -12200.539,E2 -12200.539} C_VEL
LIN {X 0,Y 375.943,Z 240.153,A -85,B 0,C 180,E1 -12203.502,E2 -12203.502} C_VEL
LIN {X 0,Y 375.943,Z 240.152,A -85,B 0,C 180,E1 -12205.893,E2 -12205.893} C_VEL
LIN {X 0,Y 375.949,Z 240.152,A -85,B 0,C 180,E1 -12209.692,E2 -12209.692} C_VEL
LIN {X 0,Y 375.907,Z 240.156,A -85,B 0,C 180,E1 -12212.14,E2 -12212.14} C_VEL
LIN {X 0,Y 375.927,Z 240.154,A -85,B 0,C 180,E1 -12214.539,E2 -12214.539} C_VEL
LIN {X 0,Y 375.965,Z 240.151,A -85,B 0,C 180,E1 -12216.892,E2 -12216.892} C_VEL
LIN {X 0,Y 375.992,Z 240.146,A -85,B 0,C 180,E1 -12220.344,E2 -12220.344} C_VEL
LIN {X 0,Y 376.023,Z 240.148,A -85,B 0,C 180,E1 -12223.724,E2 -12223.724} C_VEL
LIN {X 0,Y 376.102,Z 240.132,A -85,B 0,C 180,E1 -12227.047,E2 -12227.047} C_VEL
LIN {X 0,Y 376.11,Z 240.133,A -85,B 0,C 180,E1 -12230.323,E2 -12230.323} C_VEL
LIN {X 0,Y 376.196,Z 240.123,A -85,B 0,C 180,E1 -12233.569,E2 -12233.569} C_VEL
LIN {X 0,Y 376.344,Z 240.106,A -85,B 0,C 180,E1 -12237.864,E2 -12237.864} C_VEL
LIN {X 0,Y 376.34,Z 240.108,A -85,B 0,C 180,E1 -12242.145,E2 -12242.145} C_VEL
LIN {X 0,Y 376.203,Z 240.126,A -85,B 0,C 180,E1 -12246.44,E2 -12246.44} C_VEL
LIN {X 0,Y 376.12,Z 240.13,A -85,B 0,C 180,E1 -12249.685,E2 -12249.685} C_VEL
LIN {X 0,Y 376.103,Z 240.132,A -85,B 0,C 180,E1 -12253.661,E2 -12253.661} C_VEL
LIN {X 0,Y 376.046,Z 240.139,A -85,B 0,C 180,E1 -12257.403,E2 -12257.403} C_VEL
LIN {X 0,Y 375.994,Z 240.153,A -85,B 0,C 180,E1 -12260.835,E2 -12260.835} C_VEL
LIN {X 0,Y 375.984,Z 240.147,A -85,B 0,C 180,E1 -12264.286,E2 -12264.286} C_VEL
LIN {X 0,Y 375.933,Z 240.153,A -85,B 0,C 180,E1 -12267.867,E2 -12267.867} C_VEL
LIN {X 0,Y 375.972,Z 240.151,A -85,B 0,C 180,E1 -12271.564,E2 -12271.564} C_VEL
LIN {X 0,Y 375.972,Z 240.154,A -85,B 0,C 180,E1 -12275.417,E2 -12275.417} C_VEL
LIN {X 0,Y 375.952,Z 240.151,A -85,B 0,C 180,E1 -12278.264,E2 -12278.264} C_VEL
LIN {X 0,Y 375.93,Z 240.16,A -85,B 0,C 180,E1 -12281.598,E2 -12281.598} C_VEL
LIN {X 0,Y 375.936,Z 240.152,A -85,B 0,C 180,E1 -12284.731,E2 -12284.731} C_VEL
LIN {X 0,Y 375.924,Z 240.161,A -85,B 0,C 180,E1 -12287.697,E2 -12287.697} C_VEL
LIN {X 0,Y 375.951,Z 240.151,A -85,B 0,C 180,E1 -12290.534,E2 -12290.534} C_VEL
LIN {X 0,Y 375.979,Z 240.15,A -85,B 0,C 180,E1 -12293.496,E2 -12293.496} C_VEL
LIN {X 0,Y 375.977,Z 240.154,A -85,B 0,C 180,E1 -12295.889,E2 -12295.889} C_VEL
LIN {X 0,Y 375.978,Z 240.15,A -85,B 0,C 180,E1 -12299.687,E2 -12299.687} C_VEL
LIN {X 0,Y 376.02,Z 240.248,A -85,B 0,C 180,E1 -12302.369,E2 -12302.369} C_VEL
LIN {X 0,Y 377.519,Z 247.778,A -85,B 0,C 180,E1 -12304.351,E2 -12304.351} C_VEL
LIN {X 0,Y 378.854,Z 255.257,A -85,B 0,C 180,E1 -12306.203,E2 -12306.203} C_VEL
LIN {X 0,Y 378.449,Z 262.616,A -85,B 0,C 180,E1 -12307.909,E2 -12307.909} C_VEL
LIN {X 0,Y 377.988,Z 268.981,A -85,B 0,C 180,E1 -12309.311,E2 -12309.311} C_VEL
LIN {X 0,Y 382.556,Z 298.62,A -85,B 0,C 180,E1 -12310.141,E2 -12310.141} C_VEL
LIN {X 0,Y 381.352,Z 376.361,A -85,B 0,C 180,E1 -12311.636,E2 -12311.636} C_VEL
LIN {X 0,Y 380.801,Z 389.696,A -85,B 0,C 180,E1 -12312.096,E2 -12312.096} C_VEL
LIN {X 0,Y 380.046,Z 403.052,A -85,B 0,C 180,E1 -12312.788,E2 -12312.788} C_VEL
LIN {X 0,Y 379.272,Z 414.261,A -85,B 0,C 180,E1 -12313.584,E2 -12313.584} C_VEL
LIN {X 0,Y 378.397,Z 425.913,A -85,B 0,C 180,E1 -12314.651,E2 -12314.651} C_VEL
LIN {X 0,Y 377.605,Z 436.189,A -85,B 0,C 180,E1 -12315.832,E2 -12315.832} C_VEL
LIN {X 0,Y 376.831,Z 444.952,A -85,B 0,C 180,E1 -12317.066,E2 -12317.066} C_VEL
LIN {X 0,Y 375.948,Z 454.194,A -85,B 0,C 180,E1 -12318.678,E2 -12318.678} C_VEL
LIN {X 0,Y 375.374,Z 461.622,A -85,B 0,C 180,E1 -12320.298,E2 -12320.298} C_VEL
LIN {X 0,Y 374.918,Z 467.57,A -85,B 0,C 180,E1 -12321.916,E2 -12321.916} C_VEL
LIN {X 0,Y 374.643,Z 472.255,A -85,B 0,C 180,E1 -12323.536,E2 -12323.536} C_VEL
LIN {X 0,Y 374.554,Z 475.817,A -85,B 0,C 180,E1 -12325.155,E2 -12325.155} C_VEL
LIN {X 0,Y 374.438,Z 478.357,A -85,B 0,C 180,E1 -12326.77,E2 -12326.77} C_VEL
LIN {X 0,Y 374.42,Z 479.544,A -85,B 0,C 180,E1 -12327.847,E2 -12327.847} C_VEL
LIN {X 0,Y 374.458,Z 480.285,A -85,B 0,C 180,E1 -12328.923,E2 -12328.923} C_VEL
LIN {X 0,Y 374.479,Z 480.634,A -85,B 0,C 180,E1 -12329.998,E2 -12329.998} C_VEL
LIN {X 0,Y 374.457,Z 480.596,A -85,B 0,C 180,E1 -12331.074,E2 -12331.074} C_VEL
LIN {X 0,Y 374.418,Z 480.17,A -85,B 0,C 180,E1 -12332.15,E2 -12332.15} C_VEL
LIN {X 0,Y 374.563,Z 478.05,A -85,B 0,C 180,E1 -12334.303,E2 -12334.303} C_VEL
LIN {X 0,Y 374.651,Z 474.935,A -85,B 0,C 180,E1 -12336.148,E2 -12336.148} C_VEL
LIN {X 0,Y 375.026,Z 470.281,A -85,B 0,C 180,E1 -12338.078,E2 -12338.078} C_VEL
LIN {X 0,Y 375.608,Z 464.113,A -85,B 0,C 180,E1 -12339.965,E2 -12339.965} C_VEL
LIN {X 0,Y 376.32,Z 457.409,A -85,B 0,C 180,E1 -12341.58,E2 -12341.58} C_VEL
LIN {X 0,Y 377.394,Z 449.105,A -85,B 0,C 180,E1 -12343.185,E2 -12343.185} C_VEL
LIN {X 0,Y 378.339,Z 440.58,A -85,B 0,C 180,E1 -12344.522,E2 -12344.522} C_VEL
LIN {X 0,Y 379.393,Z 430.326,A -85,B 0,C 180,E1 -12345.827,E2 -12345.827} C_VEL
LIN {X 0,Y 380.478,Z 419.719,A -85,B 0,C 180,E1 -12346.912,E2 -12346.912} C_VEL
LIN {X 0,Y 381.557,Z 408.335,A -85,B 0,C 180,E1 -12347.83,E2 -12347.83} C_VEL
LIN {X 0,Y 382.509,Z 395.324,A -85,B 0,C 180,E1 -12348.615,E2 -12348.615} C_VEL
LIN {X 0,Y 383.283,Z 382.25,A -85,B 0,C 180,E1 -12349.166,E2 -12349.166} C_VEL
LIN {X 0,Y 383.735,Z 369.201,A -85,B 0,C 180,E1 -12349.5,E2 -12349.5} C_VEL
LIN {X 0,Y 384.9,Z 298.249,A -85,B 0,C 180,E1 -12350.872,E2 -12350.872} C_VEL
LIN {X 0,Y 381.375,Z 278.862,A -85,B 0,C 180,E1 -12351.51,E2 -12351.51} C_VEL
LIN {X 0,Y 379.165,Z 268.641,A -85,B 0,C 180,E1 -12351.908,E2 -12351.908} C_VEL
LIN {X 0,Y 379.941,Z 259.374,A -85,B 0,C 180,E1 -12354.011,E2 -12354.011} C_VEL
LIN {X 0,Y 378.204,Z 249.868,A -85,B 0,C 180,E1 -12356.484,E2 -12356.484} C_VEL
LIN {X 0,Y 376.034,Z 240.501,A -85,B 0,C 180,E1 -12359.072,E2 -12359.072} C_VEL
LIN {X 0,Y 375.975,Z 240.154,A -85,B 0,C 180,E1 -12359.383,E2 -12359.383} C_VEL
LIN {X 0,Y 375.954,Z 240.15,A -85,B 0,C 180,E1 -12362.826,E2 -12362.826} C_VEL
LIN {X 0,Y 375.961,Z 240.147,A -85,B 0,C 180,E1 -12365.413,E2 -12365.413} C_VEL
LIN {X 0,Y 375.942,Z 240.148,A -85,B 0,C 180,E1 -12368.26,E2 -12368.26} C_VEL
LIN {X 0,Y 375.925,Z 240.149,A -85,B 0,C 180,E1 -12371.595,E2 -12371.595} C_VEL
LIN {X 0,Y 375.927,Z 240.154,A -85,B 0,C 180,E1 -12375.266,E2 -12375.266} C_VEL
LIN {X 0,Y 375.919,Z 240.155,A -85,B 0,C 180,E1 -12378.399,E2 -12378.399} C_VEL
LIN {X 0,Y 375.953,Z 240.153,A -85,B 0,C 180,E1 -12381.907,E2 -12381.907} C_VEL
LIN {X 0,Y 375.979,Z 240.15,A -85,B 0,C 180,E1 -12385.329,E2 -12385.329} C_VEL
LIN {X 0,Y 375.955,Z 240.153,A -85,B 0,C 180,E1 -12388.434,E2 -12388.434} C_VEL
LIN {X 0,Y 375.926,Z 240.155,A -85,B 0,C 180,E1 -12392.132,E2 -12392.132} C_VEL
LIN {X 0,Y 375.955,Z 240.15,A -85,B 0,C 180,E1 -12395.712,E2 -12395.712} C_VEL
LIN {X 0,Y 375.974,Z 240.146,A -85,B 0,C 180,E1 -12399.193,E2 -12399.193} C_VEL
LIN {X 0,Y 376.026,Z 240.142,A -85,B 0,C 180,E1 -12402.596,E2 -12402.596} C_VEL
LIN {X 0,Y 376.082,Z 240.136,A -85,B 0,C 180,E1 -12406.339,E2 -12406.339} C_VEL
LIN {X 0,Y 376.099,Z 240.134,A -85,B 0,C 180,E1 -12410.314,E2 -12410.314} C_VEL
LIN {X 0,Y 376.206,Z 240.121,A -85,B 0,C 180,E1 -12413.56,E2 -12413.56} C_VEL
LIN {X 0,Y 376.318,Z 240.107,A -85,B 0,C 180,E1 -12417.855,E2 -12417.855} C_VEL
LIN {X 0,Y 376.323,Z 240.106,A -85,B 0,C 180,E1 -12422.136,E2 -12422.136} C_VEL
LIN {X 0,Y 376.174,Z 240.124,A -85,B 0,C 180,E1 -12426.433,E2 -12426.433} C_VEL
LIN {X 0,Y 376.094,Z 240.132,A -85,B 0,C 180,E1 -12429.678,E2 -12429.678} C_VEL
LIN {X 0,Y 376.069,Z 240.135,A -85,B 0,C 180,E1 -12433.653,E2 -12433.653} C_VEL
LIN {X 0,Y 376.009,Z 240.143,A -85,B 0,C 180,E1 -12437.396,E2 -12437.396} C_VEL
LIN {X 0,Y 375.954,Z 240.153,A -85,B 0,C 180,E1 -12440.828,E2 -12440.828} C_VEL
LIN {X 0,Y 375.961,Z 240.155,A -85,B 0,C 180,E1 -12444.278,E2 -12444.278} C_VEL
LIN {X 0,Y 375.992,Z 240.15,A -85,B 0,C 180,E1 -12446.648,E2 -12446.648} C_VEL
LIN {X 0,Y 375.935,Z 240.156,A -85,B 0,C 180,E1 -12450.309,E2 -12450.309} C_VEL
LIN {X 0,Y 375.928,Z 240.158,A -85,B 0,C 180,E1 -12454.108,E2 -12454.108} C_VEL
LIN {X 0,Y 375.923,Z 240.158,A -85,B 0,C 180,E1 -12456.738,E2 -12456.738} C_VEL
LIN {X 0,Y 375.965,Z 240.153,A -85,B 0,C 180,E1 -12459.97,E2 -12459.97} C_VEL
LIN {X 0,Y 375.998,Z 240.229,A -85,B 0,C 180,E1 -12462.091,E2 -12462.091} C_VEL
LIN {X 0,Y 377.956,Z 249.019,A -85,B 0,C 180,E1 -12464.576,E2 -12464.576} C_VEL
LIN {X 0,Y 379.424,Z 257.231,A -85,B 0,C 180,E1 -12466.74,E2 -12466.74} C_VEL
LIN {X 0,Y 379.438,Z 259.389,A -85,B 0,C 180,E1 -12467.16,E2 -12467.16} C_VEL
LIN {X 0,Y 383.907,Z 279.134,A -85,B 0,C 180,E1 -12467.908,E2 -12467.908} C_VEL
LIN {X 0,Y 385.169,Z 285.914,A -85,B 0,C 180,E1 -12468.131,E2 -12468.131} C_VEL
LIN {X 0,Y 383.601,Z 367.528,A -85,B 0,C 180,E1 -12469.732,E2 -12469.732} C_VEL
LIN {X 0,Y 382.939,Z 381.248,A -85,B 0,C 180,E1 -12470.229,E2 -12470.229} C_VEL
LIN {X 0,Y 382.176,Z 393.595,A -85,B 0,C 180,E1 -12470.897,E2 -12470.897} C_VEL
LIN {X 0,Y 381.274,Z 404.678,A -85,B 0,C 180,E1 -12471.7,E2 -12471.7} C_VEL
LIN {X 0,Y 380.188,Z 415.946,A -85,B 0,C 180,E1 -12472.745,E2 -12472.745} C_VEL
LIN {X 0,Y 379.041,Z 426.252,A -85,B 0,C 180,E1 -12473.938,E2 -12473.938} C_VEL
LIN {X 0,Y 378.106,Z 434.699,A -85,B 0,C 180,E1 -12475.143,E2 -12475.143} C_VEL
LIN {X 0,Y 377.163,Z 443.05,A -85,B 0,C 180,E1 -12476.595,E2 -12476.595} C_VEL
LIN {X 0,Y 376.285,Z 450.33,A -85,B 0,C 180,E1 -12478.157,E2 -12478.157} C_VEL
LIN {X 0,Y 375.707,Z 456.032,A -85,B 0,C 180,E1 -12479.667,E2 -12479.667} C_VEL
LIN {X 0,Y 375.212,Z 461.043,A -85,B 0,C 180,E1 -12481.332,E2 -12481.332} C_VEL
LIN {X 0,Y 374.77,Z 465.389,A -85,B 0,C 180,E1 -12483.254,E2 -12483.254} C_VEL
LIN {X 0,Y 374.555,Z 467.354,A -85,B 0,C 180,E1 -12484.435,E2 -12484.435} C_VEL
LIN {X 0,Y 374.356,Z 468.785,A -85,B 0,C 180,E1 -12485.608,E2 -12485.608} C_VEL
LIN {X 0,Y 374.251,Z 469.862,A -85,B 0,C 180,E1 -12486.934,E2 -12486.934} C_VEL
LIN {X 0,Y 374.218,Z 470.245,A -85,B 0,C 180,E1 -12487.94,E2 -12487.94} C_VEL
LIN {X 0,Y 374.24,Z 470.031,A -85,B 0,C 180,E1 -12489.861,E2 -12489.861} C_VEL
LIN {X 0,Y 374.275,Z 468.975,A -85,B 0,C 180,E1 -12491.386,E2 -12491.386} C_VEL
LIN {X 0,Y 374.455,Z 466.706,A -85,B 0,C 180,E1 -12493.154,E2 -12493.154} C_VEL
LIN {X 0,Y 374.664,Z 463.608,A -85,B 0,C 180,E1 -12494.777,E2 -12494.777} C_VEL
LIN {X 0,Y 374.998,Z 459.109,A -85,B 0,C 180,E1 -12496.509,E2 -12496.509} C_VEL
LIN {X 0,Y 375.466,Z 452.68,A -85,B 0,C 180,E1 -12498.394,E2 -12498.394} C_VEL
LIN {X 0,Y 376.024,Z 445.454,A -85,B 0,C 180,E1 -12500.046,E2 -12500.046} C_VEL
LIN {X 0,Y 376.87,Z 436.371,A -85,B 0,C 180,E1 -12501.692,E2 -12501.692} C_VEL
LIN {X 0,Y 377.627,Z 427.081,A -85,B 0,C 180,E1 -12503.054,E2 -12503.054} C_VEL
LIN {X 0,Y 378.58,Z 416.666,A -85,B 0,C 180,E1 -12504.275,E2 -12504.275} C_VEL
LIN {X 0,Y 379.47,Z 405.109,A -85,B 0,C 180,E1 -12505.354,E2 -12505.354} C_VEL
LIN {X 0,Y 380.201,Z 393.362,A -85,B 0,C 180,E1 -12506.21,E2 -12506.21} C_VEL
LIN {X 0,Y 380.861,Z 380.506,A -85,B 0,C 180,E1 -12506.894,E2 -12506.894} C_VEL
LIN {X 0,Y 381.369,Z 367.495,A -85,B 0,C 180,E1 -12507.361,E2 -12507.361} C_VEL
LIN {X 0,Y 382.146,Z 315.454,A -85,B 0,C 180,E1 -12508.383,E2 -12508.383} C_VEL
LIN {X 0,Y 382.473,Z 283.94,A -85,B 0,C 180,E1 -12508.985,E2 -12508.985} C_VEL
LIN {X 0,Y 378.249,Z 259.593,A -85,B 0,C 180,E1 -12509.687,E2 -12509.687} C_VEL
LIN {X 0,Y 378.214,Z 258.952,A -85,B 0,C 180,E1 -12509.759,E2 -12509.759} C_VEL
LIN {X 0,Y 377.894,Z 257.019,A -85,B 0,C 180,E1 -12510.222,E2 -12510.222} C_VEL
LIN {X 0,Y 375.805,Z 253.453,A -85,B 0,C 180,E1 -12511.225,E2 -12511.225} C_VEL
LIN {X 0,Y 371.476,Z 248.332,A -85,B 0,C 180,E1 -12512.801,E2 -12512.801} C_VEL
LIN {X 0,Y 369.638,Z 244.48,A -85,B 0,C 180,E1 -12513.89,E2 -12513.89} C_VEL
LIN {X 0,Y 369.054,Z 241.081,A -85,B 0,C 180,E1 -12514.883,E2 -12514.883} C_VEL
LIN {X 0,Y 369.122,Z 241.006,A -85,B 0,C 180,E1 -12517.661,E2 -12517.661} C_VEL
LIN {X 0,Y 368.988,Z 241.019,A -85,B 0,C 180,E1 -12520.982,E2 -12520.982} C_VEL
LIN {X 0,Y 368.978,Z 241.02,A -85,B 0,C 180,E1 -12524.338,E2 -12524.338} C_VEL
LIN {X 0,Y 368.966,Z 241.028,A -85,B 0,C 180,E1 -12527.772,E2 -12527.772} C_VEL
LIN {X 0,Y 368.875,Z 241.033,A -85,B 0,C 180,E1 -12531.225,E2 -12531.225} C_VEL
LIN {X 0,Y 368.888,Z 241.036,A -85,B 0,C 180,E1 -12533.882,E2 -12533.882} C_VEL
LIN {X 0,Y 368.839,Z 241.037,A -85,B 0,C 180,E1 -12537.215,E2 -12537.215} C_VEL
LIN {X 0,Y 368.864,Z 241.035,A -85,B 0,C 180,E1 -12539.696,E2 -12539.696} C_VEL
LIN {X 0,Y 368.867,Z 241.033,A -85,B 0,C 180,E1 -12543.047,E2 -12543.047} C_VEL
LIN {X 0,Y 368.883,Z 241.036,A -85,B 0,C 180,E1 -12546.202,E2 -12546.202} C_VEL
LIN {X 0,Y 368.847,Z 241.038,A -85,B 0,C 180,E1 -12548.962,E2 -12548.962} C_VEL
LIN {X 0,Y 368.834,Z 241.038,A -85,B 0,C 180,E1 -12552.01,E2 -12552.01} C_VEL
LIN {X 0,Y 368.854,Z 241.037,A -85,B 0,C 180,E1 -12555.18,E2 -12555.18} C_VEL
LIN {X 0,Y 368.85,Z 241.036,A -85,B 0,C 180,E1 -12558.181,E2 -12558.181} C_VEL
LIN {X 0,Y 368.86,Z 241.036,A -85,B 0,C 180,E1 -12561.371,E2 -12561.371} C_VEL
LIN {X 0,Y 368.916,Z 241.033,A -85,B 0,C 180,E1 -12565.151,E2 -12565.151} C_VEL
LIN {X 0,Y 368.884,Z 241.037,A -85,B 0,C 180,E1 -12569.049,E2 -12569.049} C_VEL
LIN {X 0,Y 368.897,Z 241.033,A -85,B 0,C 180,E1 -12571.563,E2 -12571.563} C_VEL
LIN {X 0,Y 368.878,Z 241.037,A -85,B 0,C 180,E1 -12575.225,E2 -12575.225} C_VEL
LIN {X 0,Y 368.913,Z 241.032,A -85,B 0,C 180,E1 -12577.609,E2 -12577.609} C_VEL
LIN {X 0,Y 368.951,Z 241.025,A -85,B 0,C 180,E1 -12581.111,E2 -12581.111} C_VEL
LIN {X 0,Y 368.994,Z 241.017,A -85,B 0,C 180,E1 -12584.54,E2 -12584.54} C_VEL
LIN {X 0,Y 369.057,Z 241.009,A -85,B 0,C 180,E1 -12586.795,E2 -12586.795} C_VEL
LIN {X 0,Y 369.06,Z 241.013,A -85,B 0,C 180,E1 -12590.136,E2 -12590.136} C_VEL
LIN {X 0,Y 369.158,Z 240.999,A -85,B 0,C 180,E1 -12593.445,E2 -12593.445} C_VEL
LIN {X 0,Y 369.307,Z 240.982,A -85,B 0,C 180,E1 -12597.823,E2 -12597.823} C_VEL
LIN {X 0,Y 369.303,Z 240.986,A -85,B 0,C 180,E1 -12602.185,E2 -12602.185} C_VEL
LIN {X 0,Y 369.164,Z 241.001,A -85,B 0,C 180,E1 -12606.563,E2 -12606.563} C_VEL
LIN {X 0,Y 369.071,Z 241.009,A -85,B 0,C 180,E1 -12609.872,E2 -12609.872} C_VEL
LIN {X 0,Y 369.051,Z 241.01,A -85,B 0,C 180,E1 -12613.775,E2 -12613.775} C_VEL
LIN {X 0,Y 369.005,Z 241.016,A -85,B 0,C 180,E1 -12617.746,E2 -12617.746} C_VEL
LIN {X 0,Y 368.924,Z 241.029,A -85,B 0,C 180,E1 -12621.224,E2 -12621.224} C_VEL
LIN {X 0,Y 368.938,Z 241.029,A -85,B 0,C 180,E1 -12624.78,E2 -12624.78} C_VEL
LIN {X 0,Y 368.909,Z 241.031,A -85,B 0,C 180,E1 -12628.794,E2 -12628.794} C_VEL
LIN {X 0,Y 368.913,Z 241.027,A -85,B 0,C 180,E1 -12632.24,E2 -12632.24} C_VEL
LIN {X 0,Y 368.944,Z 241.027,A -85,B 0,C 180,E1 -12635.003,E2 -12635.003} C_VEL
LIN {X 0,Y 368.893,Z 241.03,A -85,B 0,C 180,E1 -12638.635,E2 -12638.635} C_VEL
LIN {X 0,Y 368.875,Z 241.034,A -85,B 0,C 180,E1 -12642.006,E2 -12642.006} C_VEL
LIN {X 0,Y 368.889,Z 241.033,A -85,B 0,C 180,E1 -12645.175,E2 -12645.175} C_VEL
LIN {X 0,Y 368.877,Z 241.034,A -85,B 0,C 180,E1 -12648.175,E2 -12648.175} C_VEL
LIN {X 0,Y 368.893,Z 241.032,A -85,B 0,C 180,E1 -12651.367,E2 -12651.367} C_VEL
LIN {X 0,Y 368.953,Z 241.023,A -85,B 0,C 180,E1 -12655.147,E2 -12655.147} C_VEL
LIN {X 0,Y 368.93,Z 241.03,A -85,B 0,C 180,E1 -12659.045,E2 -12659.045} C_VEL
LIN {X 0,Y 368.976,Z 241.247,A -85,B 0,C 180,E1 -12662.181,E2 -12662.181} C_VEL
LIN {X 0,Y 370.934,Z 251.107,A -85,B 0,C 180,E1 -12664.766,E2 -12664.766} C_VEL
LIN {X 0,Y 371.94,Z 257.328,A -85,B 0,C 180,E1 -12666.325,E2 -12666.325} C_VEL
LIN {X 0,Y 371.08,Z 268.631,A -85,B 0,C 180,E1 -12668.946,E2 -12668.946} C_VEL
LIN {X 0,Y 371.692,Z 272.918,A -85,B 0,C 180,E1 -12669.121,E2 -12669.121} C_VEL
LIN {X 0,Y 375.749,Z 299.683,A -85,B 0,C 180,E1 -12669.85,E2 -12669.85} C_VEL
LIN {X 0,Y 374.514,Z 376.494,A -85,B 0,C 180,E1 -12671.36,E2 -12671.36} C_VEL
LIN {X 0,Y 373.947,Z 389.746,A -85,B 0,C 180,E1 -12671.827,E2 -12671.827} C_VEL
LIN {X 0,Y 373.17,Z 403.059,A -85,B 0,C 180,E1 -12672.532,E2 -12672.532} C_VEL
LIN {X 0,Y 372.299,Z 415.034,A -85,B 0,C 180,E1 -12673.409,E2 -12673.409} C_VEL
LIN {X 0,Y 371.397,Z 426.528,A -85,B 0,C 180,E1 -12674.495,E2 -12674.495} C_VEL
LIN {X 0,Y 370.557,Z 436.884,A -85,B 0,C 180,E1 -12675.724,E2 -12675.724} C_VEL
LIN {X 0,Y 369.714,Z 446.159,A -85,B 0,C 180,E1 -12677.092,E2 -12677.092} C_VEL
LIN {X 0,Y 368.826,Z 455.166,A -85,B 0,C 180,E1 -12678.735,E2 -12678.735} C_VEL
LIN {X 0,Y 368.241,Z 462.409,A -85,B 0,C 180,E1 -12680.385,E2 -12680.385} C_VEL
LIN {X 0,Y 367.876,Z 467.285,A -85,B 0,C 180,E1 -12681.761,E2 -12681.761} C_VEL
LIN {X 0,Y 367.576,Z 472.013,A -85,B 0,C 180,E1 -12683.411,E2 -12683.411} C_VEL
LIN {X 0,Y 367.455,Z 475.612,A -85,B 0,C 180,E1 -12685.061,E2 -12685.061} C_VEL
LIN {X 0,Y 367.358,Z 478.188,A -85,B 0,C 180,E1 -12686.708,E2 -12686.708} C_VEL
LIN {X 0,Y 367.323,Z 479.396,A -85,B 0,C 180,E1 -12687.805,E2 -12687.805} C_VEL
LIN {X 0,Y 367.357,Z 480.163,A -85,B 0,C 180,E1 -12688.902,E2 -12688.902} C_VEL
LIN {X 0,Y 367.38,Z 480.527,A -85,B 0,C 180,E1 -12689.998,E2 -12689.998} C_VEL
LIN {X 0,Y 367.356,Z 480.505,A -85,B 0,C 180,E1 -12691.094,E2 -12691.094} C_VEL
LIN {X 0,Y 367.322,Z 480.1,A -85,B 0,C 180,E1 -12692.191,E2 -12692.191} C_VEL
LIN {X 0,Y 367.36,Z 479.27,A -85,B 0,C 180,E1 -12693.288,E2 -12693.288} C_VEL
LIN {X 0,Y 367.472,Z 478.028,A -85,B 0,C 180,E1 -12694.386,E2 -12694.386} C_VEL
LIN {X 0,Y 367.55,Z 475.275,A -85,B 0,C 180,E1 -12696.1,E2 -12696.1} C_VEL
LIN {X 0,Y 367.971,Z 470.344,A -85,B 0,C 180,E1 -12698.234,E2 -12698.234} C_VEL
LIN {X 0,Y 368.616,Z 464.23,A -85,B 0,C 180,E1 -12700.156,E2 -12700.156} C_VEL
LIN {X 0,Y 369.334,Z 457.574,A -85,B 0,C 180,E1 -12701.802,E2 -12701.802} C_VEL
LIN {X 0,Y 370.495,Z 449.326,A -85,B 0,C 180,E1 -12703.435,E2 -12703.435} C_VEL
LIN {X 0,Y 371.565,Z 440.051,A -85,B 0,C 180,E1 -12704.914,E2 -12704.914} C_VEL
LIN {X 0,Y 372.67,Z 429.443,A -85,B 0,C 180,E1 -12706.275,E2 -12706.275} C_VEL
LIN {X 0,Y 373.831,Z 418.809,A -85,B 0,C 180,E1 -12707.363,E2 -12707.363} C_VEL
LIN {X 0,Y 375.028,Z 407.12,A -85,B 0,C 180,E1 -12708.292,E2 -12708.292} C_VEL
LIN {X 0,Y 375.919,Z 395.034,A -85,B 0,C 180,E1 -12709.024,E2 -12709.024} C_VEL
LIN {X 0,Y 376.719,Z 381.888,A -85,B 0,C 180,E1 -12709.584,E2 -12709.584} C_VEL
LIN {X 0,Y 377.204,Z 368.357,A -85,B 0,C 180,E1 -12709.927,E2 -12709.927} C_VEL
LIN {X 0,Y 378.381,Z 298.837,A -85,B 0,C 180,E1 -12711.298,E2 -12711.298} C_VEL
LIN {X 0,Y 374.306,Z 277.034,A -85,B 0,C 180,E1 -12712.048,E2 -12712.048} C_VEL
LIN {X 0,Y 372.38,Z 268.388,A -85,B 0,C 180,E1 -12712.416,E2 -12712.416} C_VEL
LIN {X 0,Y 373.038,Z 260.78,A -85,B 0,C 180,E1 -12714.188,E2 -12714.188} C_VEL
LIN {X 0,Y 371.013,Z 249.959,A -85,B 0,C 180,E1 -12717.083,E2 -12717.083} C_VEL
LIN {X 0,Y 368.953,Z 241.089,A -85,B 0,C 180,E1 -12719.656,E2 -12719.656} C_VEL
LIN {X 0,Y 368.902,Z 241.032,A -85,B 0,C 180,E1 -12723.535,E2 -12723.535} C_VEL
LIN {X 0,Y 368.903,Z 241.033,A -85,B 0,C 180,E1 -12726.852,E2 -12726.852} C_VEL
LIN {X 0,Y 368.91,Z 241.032,A -85,B 0,C 180,E1 -12730.368,E2 -12730.368} C_VEL
